SPLINE
SPL {X  -156.240, Y  +354.319, Z    +0.000, E1   +23.538, E3 +157736.290}
SPL {X  -159.137, Y  +372.201, Z    +0.000, E1   +12.017, E3 +157766.128}
SPL {X  -159.858, Y  +382.069, Z    +0.000, E1    +5.945, E3 +157772.645}
SPL {X  -160.000, Y  +389.339, Z    +0.000, E1    +1.101, E3 +157775.807}
SPL {X  -160.000, Y  +395.749, Z    +0.000, E1    -3.722, E3 +157778.413}
SPL {X  -160.000, Y  +403.128, Z    +0.000, E1    -9.899, E3 +157781.717}
SPL {X  -160.000, Y  +411.609, Z    +0.000, E1   -16.851, E3 +157787.038}
SPL {X  -160.000, Y  +429.715, Z    +0.000, E1   -27.376, E3 +157806.401}
SPL {X  -160.000, Y  +449.791, Z    +0.000, E1   -32.145, E3 +157847.638}
SPL {X  -160.000, Y  +454.903, Z    +0.000, E1   -32.134, E3 +157864.943}
SPL {X  -160.000, Y  +460.041, Z    +0.000, E1   -32.144, E3 +157882.296}
SPL {X  -160.000, Y  +465.466, Z    +0.000, E1   -32.152, E3 +157900.614}
SPL {X  -160.000, Y  +471.112, Z    +0.000, E1   -32.154, E3 +157919.702}
SPL {X  -160.000, Y  +476.735, Z    +0.000, E1   -32.156, E3 +157938.693}
SPL {X  -160.000, Y  +482.675, Z    +0.000, E1   -32.169, E3 +157958.742}
SPL {X  -160.000, Y  +488.008, Z    +0.000, E1   -32.144, E3 +157976.788}
SPL {X  -160.000, Y  +493.245, Z    +0.000, E1   -32.159, E3 +157994.497}
SPL {X  -160.000, Y  +498.210, Z    +0.000, E1   -32.128, E3 +158011.331}
SPL {X  -160.000, Y  +503.407, Z    +0.000, E1   -32.165, E3 +158028.835}
SPL {X  -160.000, Y  +509.142, Z    +0.000, E1   -32.157, E3 +158048.231}
SPL {X  -160.000, Y  +514.696, Z    +0.000, E1   -32.156, E3 +158067.011}
SPL {X  -160.000, Y  +520.339, Z    +0.000, E1   -32.159, E3 +158086.083}
SPL {X  -160.000, Y  +525.825, Z    +0.000, E1   -32.148, E3 +158104.647}
SPL {X  -160.000, Y  +530.379, Z    +0.000, E1   -32.130, E3 +158120.075}
SPL {X  -160.000, Y  +535.020, Z    +0.000, E1   -32.146, E3 +158135.721}
SPL {X  -160.000, Y  +540.303, Z    +0.000, E1   -32.158, E3 +158153.546}
SPL {X  -160.000, Y  +545.740, Z    +0.000, E1   -32.155, E3 +158171.939}
SPL {X  -160.000, Y  +550.807, Z    +0.000, E1   -32.147, E3 +158189.062}
SPL {X  -160.000, Y  +555.841, Z    +0.000, E1   -32.148, E3 +158206.101}
SPL {X  -160.000, Y  +561.018, Z    +0.000, E1   -32.143, E3 +158223.630}
SPL {X  -160.000, Y  +566.466, Z    +0.000, E1   -32.153, E3 +158242.048}
SPL {X  -160.000, Y  +571.733, Z    +0.000, E1   -32.135, E3 +158259.885}
SPL {X  -160.000, Y  +576.943, Z    +0.000, E1   -32.148, E3 +158277.481}
SPL {X  -160.000, Y  +582.183, Z    +0.000, E1   -32.140, E3 +158295.206}
SPL {X  -160.000, Y  +587.036, Z    +0.000, E1   -32.141, E3 +158311.577}
SPL {X  -160.000, Y  +591.785, Z    +0.000, E1   -32.144, E3 +158327.601}
SPL {X  -160.000, Y  +596.962, Z    +0.000, E1   -32.161, E3 +158345.087}
SPL {X  -160.000, Y  +601.800, Z    +0.000, E1   -32.134, E3 +158361.484}
SPL {X  -160.000, Y  +606.611, Z    +0.000, E1   -32.156, E3 +158377.699}
SPL {X  -160.000, Y  +611.219, Z    +0.000, E1   -32.131, E3 +158393.312}
SPL {X  -160.000, Y  +616.331, Z    +0.000, E1   -32.174, E3 +158410.510}
SPL {X  -160.000, Y  +621.751, Z    +0.000, E1   -32.150, E3 +158428.853}
SPL {X  -160.000, Y  +626.312, Z    +0.000, E1   -32.145, E3 +158444.258}
SPL {X  -160.000, Y  +630.971, Z    +0.000, E1   -32.155, E3 +158459.987}
SPL {X  -160.000, Y  +635.550, Z    +0.000, E1   -32.137, E3 +158475.513}
SPL {X  -160.000, Y  +640.419, Z    +0.000, E1   -32.158, E3 +158491.951}
SPL {X  -160.000, Y  +645.749, Z    +0.000, E1   -32.151, E3 +158509.976}
SPL {X  -160.000, Y  +650.662, Z    +0.000, E1   -32.150, E3 +158526.547}
SPL {X  -160.000, Y  +655.372, Z    +0.000, E1   -32.145, E3 +158542.494}
SPL {X  -160.000, Y  +660.593, Z    +0.000, E1   -32.163, E3 +158560.112}
SPL {X  -160.000, Y  +665.836, Z    +0.000, E1   -32.154, E3 +158577.828}
SPL {X  -160.000, Y  +670.613, Z    +0.000, E1   -32.138, E3 +158594.039}
SPL {X  -159.954, Y  +675.336, Z    +0.000, E1   -32.135, E3 +158610.047}
SPL {X  -159.758, Y  +680.302, Z    +0.000, E1   -32.108, E3 +158627.062}
SPL {X  -159.416, Y  +685.158, Z    +0.000, E1   -32.039, E3 +158643.873}
SPL {X  -158.953, Y  +689.772, Z    +0.000, E1   -31.965, E3 +158659.972}
SPL {X  -158.363, Y  +694.328, Z    +0.000, E1   -31.871, E3 +158675.985}
SPL {X  -157.606, Y  +699.074, Z    +0.000, E1   -31.756, E3 +158692.828}
SPL {X  -156.791, Y  +703.384, Z    +0.000, E1   -31.607, E3 +158708.278}
SPL {X  -155.792, Y  +707.952, Z    +0.000, E1   -31.465, E3 +158724.725}
SPL {X  -155.149, Y  +710.598, Z    +0.000, E1   -26.183, E3 +158780.185}
ENDSPLINE

SPLINE
SPL {X  -158.679, Y  +692.020, Z    +0.000, E1   -14.212, E3 +158813.861}
SPL {X  -159.747, Y  +680.500, Z    +0.000, E1    -7.378, E3 +158822.238}
SPL {X  -160.000, Y  +671.618, Z    +0.000, E1    -1.592, E3 +158825.853}
SPL {X  -160.000, Y  +666.041, Z    +0.000, E1    +2.615, E3 +158827.819}
SPL {X  -160.000, Y  +661.396, Z    +0.000, E1    +6.484, E3 +158829.492}
SPL {X  -160.000, Y  +653.532, Z    +0.000, E1   +13.136, E3 +158833.613}
SPL {X  -160.000, Y  +631.927, Z    +0.000, E1   +26.832, E3 +158856.379}
SPL {X  -160.000, Y  +610.736, Z    +0.000, E1   +32.114, E3 +158899.049}
SPL {X  -160.000, Y  +605.907, Z    +0.000, E1   +32.114, E3 +158915.397}
SPL {X  -160.000, Y  +601.221, Z    +0.000, E1   +32.108, E3 +158931.264}
SPL {X  -160.000, Y  +596.433, Z    +0.000, E1   +32.120, E3 +158947.447}
SPL {X  -160.000, Y  +592.025, Z    +0.000, E1   +32.104, E3 +158962.371}
SPL {X  -160.000, Y  +587.734, Z    +0.000, E1   +32.110, E3 +158976.891}
SPL {X  -160.000, Y  +583.150, Z    +0.000, E1   +32.111, E3 +158992.419}
SPL {X  -160.000, Y  +579.063, Z    +0.000, E1   +32.085, E3 +159006.320}
SPL {X  -160.000, Y  +574.897, Z    +0.000, E1   +32.110, E3 +159020.372}
SPL {X  -160.000, Y  +570.471, Z    +0.000, E1   +32.093, E3 +159035.386}
SPL {X  -160.000, Y  +566.667, Z    +0.000, E1   +32.086, E3 +159048.300}
SPL {X  -160.000, Y  +562.434, Z    +0.000, E1   +32.097, E3 +159062.610}
SPL {X  -160.000, Y  +557.710, Z    +0.000, E1   +32.104, E3 +159078.593}
SPL {X  -160.000, Y  +553.479, Z    +0.000, E1   +32.081, E3 +159092.963}
SPL {X  -160.000, Y  +547.489, Z    +0.000, E1   +32.181, E3 +159113.081}
SPL {X  -160.000, Y  +541.554, Z    +0.000, E1   +32.092, E3 +159133.318}
SPL {X  -160.000, Y  +537.332, Z    +0.000, E1   +32.092, E3 +159147.616}
SPL {X  -160.000, Y  +533.113, Z    +0.000, E1   +32.090, E3 +159161.912}
SPL {X  -160.000, Y  +528.875, Z    +0.000, E1   +32.090, E3 +159176.256}
SPL {X  -160.000, Y  +524.453, Z    +0.000, E1   +32.104, E3 +159191.180}
SPL {X  -160.000, Y  +520.037, Z    +0.000, E1   +32.096, E3 +159206.122}
SPL {X  -160.000, Y  +514.030, Z    +0.000, E1   +32.182, E3 +159226.318}
SPL {X  -160.000, Y  +508.131, Z    +0.000, E1   +32.099, E3 +159246.422}
SPL {X  -160.000, Y  +504.077, Z    +0.000, E1   +32.094, E3 +159260.145}
SPL {X  -160.000, Y  +494.657, Z    +0.000, E1   +34.509, E3 +159275.008}
SPL {X  -160.000, Y  +491.565, Z    +0.000, E1   +33.823, E3 +159288.915}
SPL {X  -160.000, Y  +489.317, Z    +0.000, E1   +32.894, E3 +159302.260}
SPL {X  -160.000, Y  +486.958, Z    +0.000, E1   +31.703, E3 +159318.032}
SPL {X  -160.000, Y  +484.144, Z    +0.000, E1   +30.999, E3 +159332.455}
SPL {X  -160.000, Y  +479.156, Z    +0.000, E1   +31.035, E3 +159350.021}
SPL {X  -160.000, Y  +474.045, Z    +0.000, E1   +31.015, E3 +159368.112}
SPL {X  -160.000, Y  +468.999, Z    +0.000, E1   +31.021, E3 +159385.937}
SPL {X  -160.000, Y  +464.107, Z    +0.000, E1   +31.012, E3 +159403.238}
SPL {X  -160.000, Y  +459.262, Z    +0.000, E1   +31.016, E3 +159420.345}
SPL {X  -160.000, Y  +454.119, Z    +0.000, E1   +31.026, E3 +159438.494}
SPL {X  -160.000, Y  +448.874, Z    +0.000, E1   +31.019, E3 +159457.050}
SPL {X  -160.000, Y  +443.892, Z    +0.000, E1   +31.019, E3 +159474.638}
SPL {X  -160.000, Y  +438.782, Z    +0.000, E1   +31.022, E3 +159492.712}
SPL {X  -160.000, Y  +433.722, Z    +0.000, E1   +31.007, E3 +159510.656}
SPL {X  -160.000, Y  +428.980, Z    +0.000, E1   +31.004, E3 +159527.413}
SPL {X  -160.000, Y  +424.339, Z    +0.000, E1   +31.006, E3 +159543.788}
SPL {X  -160.000, Y  +419.231, Z    +0.000, E1   +31.030, E3 +159561.781}
SPL {X  -160.000, Y  +414.179, Z    +0.000, E1   +31.008, E3 +159579.678}
SPL {X  -160.000, Y  +409.416, Z    +0.000, E1   +31.023, E3 +159596.462}
SPL {X  -160.000, Y  +403.994, Z    +0.000, E1   +31.033, E3 +159615.617}
SPL {X  -160.000, Y  +399.052, Z    +0.000, E1   +31.010, E3 +159633.085}
SPL {X  -160.000, Y  +394.012, Z    +0.000, E1   +31.036, E3 +159650.874}
SPL {X  -159.999, Y  +388.376, Z    +0.000, E1   +31.028, E3 +159670.804}
SPL {X  -159.897, Y  +383.070, Z    +0.000, E1   +31.010, E3 +159689.642}
SPL {X  -159.656, Y  +378.313, Z    +0.000, E1   +30.961, E3 +159706.734}
SPL {X  -159.237, Y  +373.190, Z    +0.000, E1   +30.917, E3 +159725.234}
SPL {X  -158.628, Y  +367.891, Z    +0.000, E1   +30.812, E3 +159744.620}
SPL {X  -157.915, Y  +363.053, Z    +0.000, E1   +30.689, E3 +159762.487}
SPL {X  -157.216, Y  +359.084, Z    +0.000, E1   +30.550, E3 +159777.289}
SPL {X  -156.248, Y  +354.355, Z    +0.000, E1   +30.460, E3 +159794.902}
SPL {X  -155.629, Y  +351.657, Z    +0.000, E1   +25.972, E3 +159841.330}
ENDSPLINE

SPLINE
SPL {X  -156.240, Y  +354.319, Z    +0.000, E1   +23.538, E3 +159853.938}
SPL {X  -159.137, Y  +372.201, Z    +0.000, E1   +12.017, E3 +159883.775}
SPL {X  -159.858, Y  +382.069, Z    +0.000, E1    +5.945, E3 +159890.293}
SPL {X  -160.000, Y  +389.339, Z    +0.000, E1    +1.101, E3 +159893.455}
SPL {X  -160.000, Y  +395.749, Z    +0.000, E1    -3.722, E3 +159896.060}
SPL {X  -160.000, Y  +403.128, Z    +0.000, E1    -9.899, E3 +159899.364}
SPL {X  -160.000, Y  +411.609, Z    +0.000, E1   -16.851, E3 +159904.685}
SPL {X  -160.000, Y  +429.715, Z    +0.000, E1   -27.376, E3 +159924.049}
SPL {X  -160.000, Y  +449.791, Z    +0.000, E1   -32.145, E3 +159965.286}
SPL {X  -160.000, Y  +454.903, Z    +0.000, E1   -32.134, E3 +159982.590}
SPL {X  -160.000, Y  +460.041, Z    +0.000, E1   -32.144, E3 +159999.943}
SPL {X  -160.000, Y  +465.466, Z    +0.000, E1   -32.152, E3 +160018.261}
SPL {X  -160.000, Y  +471.112, Z    +0.000, E1   -32.154, E3 +160037.350}
SPL {X  -160.000, Y  +476.735, Z    +0.000, E1   -32.156, E3 +160056.340}
SPL {X  -160.000, Y  +482.675, Z    +0.000, E1   -32.169, E3 +160076.389}
SPL {X  -160.000, Y  +488.008, Z    +0.000, E1   -32.144, E3 +160094.436}
SPL {X  -160.000, Y  +493.245, Z    +0.000, E1   -32.159, E3 +160112.144}
SPL {X  -160.000, Y  +498.210, Z    +0.000, E1   -32.128, E3 +160128.979}
SPL {X  -160.000, Y  +503.407, Z    +0.000, E1   -32.165, E3 +160146.482}
SPL {X  -160.000, Y  +509.142, Z    +0.000, E1   -32.157, E3 +160165.878}
SPL {X  -160.000, Y  +514.696, Z    +0.000, E1   -32.156, E3 +160184.658}
SPL {X  -160.000, Y  +520.339, Z    +0.000, E1   -32.159, E3 +160203.731}
SPL {X  -160.000, Y  +525.825, Z    +0.000, E1   -32.148, E3 +160222.294}
SPL {X  -160.000, Y  +530.379, Z    +0.000, E1   -32.130, E3 +160237.722}
SPL {X  -160.000, Y  +535.020, Z    +0.000, E1   -32.146, E3 +160253.368}
SPL {X  -160.000, Y  +540.303, Z    +0.000, E1   -32.158, E3 +160271.194}
SPL {X  -160.000, Y  +545.740, Z    +0.000, E1   -32.155, E3 +160289.586}
SPL {X  -160.000, Y  +550.807, Z    +0.000, E1   -32.147, E3 +160306.709}
SPL {X  -160.000, Y  +555.841, Z    +0.000, E1   -32.148, E3 +160323.748}
SPL {X  -160.000, Y  +561.018, Z    +0.000, E1   -32.143, E3 +160341.277}
SPL {X  -160.000, Y  +566.466, Z    +0.000, E1   -32.153, E3 +160359.695}
SPL {X  -160.000, Y  +571.733, Z    +0.000, E1   -32.135, E3 +160377.532}
SPL {X  -160.000, Y  +576.943, Z    +0.000, E1   -32.148, E3 +160395.129}
SPL {X  -160.000, Y  +582.183, Z    +0.000, E1   -32.140, E3 +160412.854}
SPL {X  -160.000, Y  +587.036, Z    +0.000, E1   -32.141, E3 +160429.224}
SPL {X  -160.000, Y  +591.785, Z    +0.000, E1   -32.144, E3 +160445.248}
SPL {X  -160.000, Y  +596.962, Z    +0.000, E1   -32.161, E3 +160462.735}
SPL {X  -160.000, Y  +601.800, Z    +0.000, E1   -32.134, E3 +160479.132}
SPL {X  -160.000, Y  +606.611, Z    +0.000, E1   -32.156, E3 +160495.346}
SPL {X  -160.000, Y  +611.219, Z    +0.000, E1   -32.131, E3 +160510.960}
SPL {X  -160.000, Y  +616.331, Z    +0.000, E1   -32.174, E3 +160528.157}
SPL {X  -160.000, Y  +621.751, Z    +0.000, E1   -32.150, E3 +160546.500}
SPL {X  -160.000, Y  +626.312, Z    +0.000, E1   -32.145, E3 +160561.906}
SPL {X  -160.000, Y  +630.971, Z    +0.000, E1   -32.155, E3 +160577.634}
SPL {X  -160.000, Y  +635.550, Z    +0.000, E1   -32.137, E3 +160593.160}
SPL {X  -160.000, Y  +640.419, Z    +0.000, E1   -32.158, E3 +160609.598}
SPL {X  -160.000, Y  +645.749, Z    +0.000, E1   -32.151, E3 +160627.623}
SPL {X  -160.000, Y  +650.662, Z    +0.000, E1   -32.150, E3 +160644.194}
SPL {X  -160.000, Y  +655.372, Z    +0.000, E1   -32.145, E3 +160660.141}
SPL {X  -160.000, Y  +660.593, Z    +0.000, E1   -32.163, E3 +160677.759}
SPL {X  -160.000, Y  +665.836, Z    +0.000, E1   -32.154, E3 +160695.476}
SPL {X  -160.000, Y  +670.613, Z    +0.000, E1   -32.138, E3 +160711.686}
SPL {X  -159.954, Y  +675.336, Z    +0.000, E1   -32.135, E3 +160727.694}
SPL {X  -159.758, Y  +680.302, Z    +0.000, E1   -32.108, E3 +160744.709}
SPL {X  -159.416, Y  +685.158, Z    +0.000, E1   -32.039, E3 +160761.520}
SPL {X  -158.953, Y  +689.772, Z    +0.000, E1   -31.965, E3 +160777.619}
SPL {X  -158.363, Y  +694.328, Z    +0.000, E1   -31.871, E3 +160793.632}
SPL {X  -157.606, Y  +699.074, Z    +0.000, E1   -31.756, E3 +160810.475}
SPL {X  -156.791, Y  +703.384, Z    +0.000, E1   -31.607, E3 +160825.926}
SPL {X  -155.792, Y  +707.952, Z    +0.000, E1   -31.465, E3 +160842.372}
SPL {X  -155.149, Y  +710.598, Z    +0.000, E1   -26.183, E3 +160897.832}
ENDSPLINE

SPLINE
SPL {X  -158.679, Y  +692.020, Z    +0.000, E1   -14.212, E3 +160931.508}
SPL {X  -159.747, Y  +680.500, Z    +0.000, E1    -7.378, E3 +160939.886}
SPL {X  -160.000, Y  +671.618, Z    +0.000, E1    -1.592, E3 +160943.500}
SPL {X  -160.000, Y  +666.041, Z    +0.000, E1    +2.615, E3 +160945.467}
SPL {X  -160.000, Y  +661.396, Z    +0.000, E1    +6.484, E3 +160947.140}
SPL {X  -160.000, Y  +653.532, Z    +0.000, E1   +13.136, E3 +160951.260}
SPL {X  -160.000, Y  +631.927, Z    +0.000, E1   +26.832, E3 +160974.027}
SPL {X  -160.000, Y  +610.736, Z    +0.000, E1   +32.114, E3 +161016.696}
SPL {X  -160.000, Y  +605.907, Z    +0.000, E1   +32.114, E3 +161033.044}
SPL {X  -160.000, Y  +601.221, Z    +0.000, E1   +32.108, E3 +161048.912}
SPL {X  -160.000, Y  +596.433, Z    +0.000, E1   +32.120, E3 +161065.094}
SPL {X  -160.000, Y  +592.025, Z    +0.000, E1   +32.104, E3 +161080.018}
SPL {X  -160.000, Y  +587.734, Z    +0.000, E1   +32.110, E3 +161094.539}
SPL {X  -160.000, Y  +583.150, Z    +0.000, E1   +32.111, E3 +161110.066}
SPL {X  -160.000, Y  +579.063, Z    +0.000, E1   +32.085, E3 +161123.968}
SPL {X  -160.000, Y  +574.897, Z    +0.000, E1   +32.110, E3 +161138.019}
SPL {X  -160.000, Y  +570.471, Z    +0.000, E1   +32.093, E3 +161153.033}
SPL {X  -160.000, Y  +566.667, Z    +0.000, E1   +32.086, E3 +161165.948}
SPL {X  -160.000, Y  +562.434, Z    +0.000, E1   +32.097, E3 +161180.257}
SPL {X  -160.000, Y  +557.710, Z    +0.000, E1   +32.104, E3 +161196.241}
SPL {X  -160.000, Y  +553.479, Z    +0.000, E1   +32.081, E3 +161210.610}
SPL {X  -160.000, Y  +547.489, Z    +0.000, E1   +32.181, E3 +161230.729}
SPL {X  -160.000, Y  +541.554, Z    +0.000, E1   +32.092, E3 +161250.966}
SPL {X  -160.000, Y  +537.332, Z    +0.000, E1   +32.092, E3 +161265.263}
SPL {X  -160.000, Y  +533.113, Z    +0.000, E1   +32.090, E3 +161279.560}
SPL {X  -160.000, Y  +528.875, Z    +0.000, E1   +32.090, E3 +161293.903}
SPL {X  -160.000, Y  +524.453, Z    +0.000, E1   +32.104, E3 +161308.827}
SPL {X  -160.000, Y  +520.037, Z    +0.000, E1   +32.096, E3 +161323.769}
SPL {X  -160.000, Y  +514.030, Z    +0.000, E1   +32.182, E3 +161343.965}
SPL {X  -160.000, Y  +508.131, Z    +0.000, E1   +32.099, E3 +161364.069}
SPL {X  -160.000, Y  +504.077, Z    +0.000, E1   +32.094, E3 +161377.792}
SPL {X  -160.000, Y  +494.657, Z    +0.000, E1   +34.509, E3 +161392.655}
SPL {X  -160.000, Y  +491.565, Z    +0.000, E1   +33.823, E3 +161406.563}
SPL {X  -160.000, Y  +489.317, Z    +0.000, E1   +32.894, E3 +161419.907}
SPL {X  -160.000, Y  +486.958, Z    +0.000, E1   +31.703, E3 +161435.679}
SPL {X  -160.000, Y  +484.144, Z    +0.000, E1   +30.999, E3 +161450.102}
SPL {X  -160.000, Y  +479.156, Z    +0.000, E1   +31.035, E3 +161467.668}
SPL {X  -160.000, Y  +474.045, Z    +0.000, E1   +31.015, E3 +161485.760}
SPL {X  -160.000, Y  +468.999, Z    +0.000, E1   +31.021, E3 +161503.585}
SPL {X  -160.000, Y  +464.107, Z    +0.000, E1   +31.012, E3 +161520.885}
SPL {X  -160.000, Y  +459.262, Z    +0.000, E1   +31.016, E3 +161537.992}
SPL {X  -160.000, Y  +454.119, Z    +0.000, E1   +31.026, E3 +161556.141}
SPL {X  -160.000, Y  +448.874, Z    +0.000, E1   +31.019, E3 +161574.697}
SPL {X  -160.000, Y  +443.892, Z    +0.000, E1   +31.019, E3 +161592.285}
SPL {X  -160.000, Y  +438.782, Z    +0.000, E1   +31.022, E3 +161610.360}
SPL {X  -160.000, Y  +433.722, Z    +0.000, E1   +31.007, E3 +161628.303}
SPL {X  -160.000, Y  +428.980, Z    +0.000, E1   +31.004, E3 +161645.061}
SPL {X  -160.000, Y  +424.339, Z    +0.000, E1   +31.006, E3 +161661.435}
SPL {X  -160.000, Y  +419.231, Z    +0.000, E1   +31.030, E3 +161679.428}
SPL {X  -160.000, Y  +414.179, Z    +0.000, E1   +31.008, E3 +161697.326}
SPL {X  -160.000, Y  +409.416, Z    +0.000, E1   +31.023, E3 +161714.109}
SPL {X  -160.000, Y  +403.994, Z    +0.000, E1   +31.033, E3 +161733.264}
SPL {X  -160.000, Y  +399.052, Z    +0.000, E1   +31.010, E3 +161750.732}
SPL {X  -160.000, Y  +394.012, Z    +0.000, E1   +31.036, E3 +161768.521}
SPL {X  -159.999, Y  +388.376, Z    +0.000, E1   +31.028, E3 +161788.451}
SPL {X  -159.897, Y  +383.070, Z    +0.000, E1   +31.010, E3 +161807.289}
SPL {X  -159.656, Y  +378.313, Z    +0.000, E1   +30.961, E3 +161824.381}
SPL {X  -159.237, Y  +373.190, Z    +0.000, E1   +30.917, E3 +161842.881}
SPL {X  -158.628, Y  +367.891, Z    +0.000, E1   +30.812, E3 +161862.267}
SPL {X  -157.915, Y  +363.053, Z    +0.000, E1   +30.689, E3 +161880.134}
SPL {X  -157.216, Y  +359.084, Z    +0.000, E1   +30.550, E3 +161894.937}
SPL {X  -156.248, Y  +354.355, Z    +0.000, E1   +30.460, E3 +161912.549}
SPL {X  -155.629, Y  +351.657, Z    +0.000, E1   +25.972, E3 +161958.977}
ENDSPLINE

SPLINE
SPL {X  -156.240, Y  +354.319, Z    +0.000, E1   +23.538, E3 +161971.585}
SPL {X  -159.137, Y  +372.201, Z    +0.000, E1   +12.017, E3 +162001.422}
SPL {X  -159.858, Y  +382.069, Z    +0.000, E1    +5.945, E3 +162007.940}
SPL {X  -160.000, Y  +389.339, Z    +0.000, E1    +1.101, E3 +162011.102}
SPL {X  -160.000, Y  +395.749, Z    +0.000, E1    -3.722, E3 +162013.707}
SPL {X  -160.000, Y  +403.128, Z    +0.000, E1    -9.899, E3 +162017.012}
SPL {X  -160.000, Y  +411.609, Z    +0.000, E1   -16.851, E3 +162022.332}
SPL {X  -160.000, Y  +429.715, Z    +0.000, E1   -27.376, E3 +162041.696}
SPL {X  -160.000, Y  +449.791, Z    +0.000, E1   -32.145, E3 +162082.933}
SPL {X  -160.000, Y  +454.903, Z    +0.000, E1   -32.134, E3 +162100.237}
SPL {X  -160.000, Y  +460.041, Z    +0.000, E1   -32.144, E3 +162117.591}
SPL {X  -160.000, Y  +465.466, Z    +0.000, E1   -32.152, E3 +162135.909}
SPL {X  -160.000, Y  +471.112, Z    +0.000, E1   -32.154, E3 +162154.997}
SPL {X  -160.000, Y  +476.735, Z    +0.000, E1   -32.156, E3 +162173.988}
SPL {X  -160.000, Y  +482.675, Z    +0.000, E1   -32.169, E3 +162194.037}
SPL {X  -160.000, Y  +488.008, Z    +0.000, E1   -32.144, E3 +162212.083}
SPL {X  -160.000, Y  +493.245, Z    +0.000, E1   -32.159, E3 +162229.791}
SPL {X  -160.000, Y  +498.210, Z    +0.000, E1   -32.128, E3 +162246.626}
SPL {X  -160.000, Y  +503.407, Z    +0.000, E1   -32.165, E3 +162264.130}
SPL {X  -160.000, Y  +509.142, Z    +0.000, E1   -32.157, E3 +162283.525}
SPL {X  -160.000, Y  +514.696, Z    +0.000, E1   -32.156, E3 +162302.306}
SPL {X  -160.000, Y  +520.339, Z    +0.000, E1   -32.159, E3 +162321.378}
SPL {X  -160.000, Y  +525.825, Z    +0.000, E1   -32.148, E3 +162339.941}
SPL {X  -160.000, Y  +530.379, Z    +0.000, E1   -32.130, E3 +162355.370}
SPL {X  -160.000, Y  +535.020, Z    +0.000, E1   -32.146, E3 +162371.016}
SPL {X  -160.000, Y  +540.303, Z    +0.000, E1   -32.158, E3 +162388.841}
SPL {X  -160.000, Y  +545.740, Z    +0.000, E1   -32.155, E3 +162407.234}
SPL {X  -160.000, Y  +550.807, Z    +0.000, E1   -32.147, E3 +162424.356}
SPL {X  -160.000, Y  +555.841, Z    +0.000, E1   -32.148, E3 +162441.396}
SPL {X  -160.000, Y  +561.018, Z    +0.000, E1   -32.143, E3 +162458.924}
SPL {X  -160.000, Y  +566.466, Z    +0.000, E1   -32.153, E3 +162477.343}
SPL {X  -160.000, Y  +571.733, Z    +0.000, E1   -32.135, E3 +162495.179}
SPL {X  -160.000, Y  +576.943, Z    +0.000, E1   -32.148, E3 +162512.776}
SPL {X  -160.000, Y  +582.183, Z    +0.000, E1   -32.140, E3 +162530.501}
SPL {X  -160.000, Y  +587.036, Z    +0.000, E1   -32.141, E3 +162546.872}
SPL {X  -160.000, Y  +591.785, Z    +0.000, E1   -32.144, E3 +162562.895}
SPL {X  -160.000, Y  +596.962, Z    +0.000, E1   -32.161, E3 +162580.382}
SPL {X  -160.000, Y  +601.800, Z    +0.000, E1   -32.134, E3 +162596.779}
SPL {X  -160.000, Y  +606.611, Z    +0.000, E1   -32.156, E3 +162612.993}
SPL {X  -160.000, Y  +611.219, Z    +0.000, E1   -32.131, E3 +162628.607}
SPL {X  -160.000, Y  +616.331, Z    +0.000, E1   -32.174, E3 +162645.805}
SPL {X  -160.000, Y  +621.751, Z    +0.000, E1   -32.150, E3 +162664.147}
SPL {X  -160.000, Y  +626.312, Z    +0.000, E1   -32.145, E3 +162679.553}
SPL {X  -160.000, Y  +630.971, Z    +0.000, E1   -32.155, E3 +162695.281}
SPL {X  -160.000, Y  +635.550, Z    +0.000, E1   -32.137, E3 +162710.807}
SPL {X  -160.000, Y  +640.419, Z    +0.000, E1   -32.158, E3 +162727.245}
SPL {X  -160.000, Y  +645.749, Z    +0.000, E1   -32.151, E3 +162745.271}
SPL {X  -160.000, Y  +650.662, Z    +0.000, E1   -32.150, E3 +162761.842}
SPL {X  -160.000, Y  +655.372, Z    +0.000, E1   -32.145, E3 +162777.789}
SPL {X  -160.000, Y  +660.593, Z    +0.000, E1   -32.163, E3 +162795.406}
SPL {X  -160.000, Y  +665.836, Z    +0.000, E1   -32.154, E3 +162813.123}
SPL {X  -160.000, Y  +670.613, Z    +0.000, E1   -32.138, E3 +162829.333}
SPL {X  -159.954, Y  +675.336, Z    +0.000, E1   -32.135, E3 +162845.341}
SPL {X  -159.758, Y  +680.302, Z    +0.000, E1   -32.108, E3 +162862.356}
SPL {X  -159.416, Y  +685.158, Z    +0.000, E1   -32.039, E3 +162879.167}
SPL {X  -158.953, Y  +689.772, Z    +0.000, E1   -31.965, E3 +162895.267}
SPL {X  -158.363, Y  +694.328, Z    +0.000, E1   -31.871, E3 +162911.279}
SPL {X  -157.606, Y  +699.074, Z    +0.000, E1   -31.756, E3 +162928.123}
SPL {X  -156.791, Y  +703.384, Z    +0.000, E1   -31.607, E3 +162943.573}
SPL {X  -155.792, Y  +707.952, Z    +0.000, E1   -31.465, E3 +162960.019}
SPL {X  -155.149, Y  +710.598, Z    +0.000, E1   -26.183, E3 +163015.479}
ENDSPLINE

SPLINE
SPL {X  -158.679, Y  +692.020, Z    +0.000, E1   -14.212, E3 +163049.155}
SPL {X  -159.747, Y  +680.500, Z    +0.000, E1    -7.378, E3 +163057.533}
SPL {X  -160.000, Y  +671.618, Z    +0.000, E1    -1.592, E3 +163061.147}
SPL {X  -160.000, Y  +666.041, Z    +0.000, E1    +2.615, E3 +163063.114}
SPL {X  -160.000, Y  +661.396, Z    +0.000, E1    +6.484, E3 +163064.787}
SPL {X  -160.000, Y  +653.532, Z    +0.000, E1   +13.136, E3 +163068.907}
SPL {X  -160.000, Y  +631.927, Z    +0.000, E1   +26.832, E3 +163091.674}
SPL {X  -160.000, Y  +610.736, Z    +0.000, E1   +32.114, E3 +163134.343}
SPL {X  -160.000, Y  +605.907, Z    +0.000, E1   +32.114, E3 +163150.692}
SPL {X  -160.000, Y  +601.221, Z    +0.000, E1   +32.108, E3 +163166.559}
SPL {X  -160.000, Y  +596.433, Z    +0.000, E1   +32.120, E3 +163182.741}
SPL {X  -160.000, Y  +592.025, Z    +0.000, E1   +32.104, E3 +163197.666}
SPL {X  -160.000, Y  +587.734, Z    +0.000, E1   +32.110, E3 +163212.186}
SPL {X  -160.000, Y  +583.150, Z    +0.000, E1   +32.111, E3 +163227.714}
SPL {X  -160.000, Y  +579.063, Z    +0.000, E1   +32.085, E3 +163241.615}
SPL {X  -160.000, Y  +574.897, Z    +0.000, E1   +32.110, E3 +163255.666}
SPL {X  -160.000, Y  +570.471, Z    +0.000, E1   +32.093, E3 +163270.681}
SPL {X  -160.000, Y  +566.667, Z    +0.000, E1   +32.086, E3 +163283.595}
SPL {X  -160.000, Y  +562.434, Z    +0.000, E1   +32.097, E3 +163297.905}
SPL {X  -160.000, Y  +557.710, Z    +0.000, E1   +32.104, E3 +163313.888}
SPL {X  -160.000, Y  +553.479, Z    +0.000, E1   +32.081, E3 +163328.257}
SPL {X  -160.000, Y  +547.489, Z    +0.000, E1   +32.181, E3 +163348.376}
SPL {X  -160.000, Y  +541.554, Z    +0.000, E1   +32.092, E3 +163368.613}
SPL {X  -160.000, Y  +537.332, Z    +0.000, E1   +32.092, E3 +163382.910}
SPL {X  -160.000, Y  +533.113, Z    +0.000, E1   +32.090, E3 +163397.207}
SPL {X  -160.000, Y  +528.875, Z    +0.000, E1   +32.090, E3 +163411.550}
SPL {X  -160.000, Y  +524.453, Z    +0.000, E1   +32.104, E3 +163426.474}
SPL {X  -160.000, Y  +520.037, Z    +0.000, E1   +32.096, E3 +163441.416}
SPL {X  -160.000, Y  +514.030, Z    +0.000, E1   +32.182, E3 +163461.612}
SPL {X  -160.000, Y  +508.131, Z    +0.000, E1   +32.099, E3 +163481.717}
SPL {X  -160.000, Y  +504.077, Z    +0.000, E1   +32.094, E3 +163495.440}
SPL {X  -160.000, Y  +494.657, Z    +0.000, E1   +34.509, E3 +163510.303}
SPL {X  -160.000, Y  +491.565, Z    +0.000, E1   +33.823, E3 +163524.210}
SPL {X  -160.000, Y  +489.317, Z    +0.000, E1   +32.894, E3 +163537.555}
SPL {X  -160.000, Y  +486.958, Z    +0.000, E1   +31.703, E3 +163553.326}
SPL {X  -160.000, Y  +484.144, Z    +0.000, E1   +30.999, E3 +163567.749}
SPL {X  -160.000, Y  +479.156, Z    +0.000, E1   +31.035, E3 +163585.315}
SPL {X  -160.000, Y  +474.045, Z    +0.000, E1   +31.015, E3 +163603.407}
SPL {X  -160.000, Y  +468.999, Z    +0.000, E1   +31.021, E3 +163621.232}
SPL {X  -160.000, Y  +464.107, Z    +0.000, E1   +31.012, E3 +163638.532}
SPL {X  -160.000, Y  +459.262, Z    +0.000, E1   +31.016, E3 +163655.639}
SPL {X  -160.000, Y  +454.119, Z    +0.000, E1   +31.026, E3 +163673.789}
SPL {X  -160.000, Y  +448.874, Z    +0.000, E1   +31.019, E3 +163692.344}
SPL {X  -160.000, Y  +443.892, Z    +0.000, E1   +31.019, E3 +163709.933}
SPL {X  -160.000, Y  +438.782, Z    +0.000, E1   +31.022, E3 +163728.007}
SPL {X  -160.000, Y  +433.722, Z    +0.000, E1   +31.007, E3 +163745.951}
SPL {X  -160.000, Y  +428.980, Z    +0.000, E1   +31.004, E3 +163762.708}
SPL {X  -160.000, Y  +424.339, Z    +0.000, E1   +31.006, E3 +163779.082}
SPL {X  -160.000, Y  +419.231, Z    +0.000, E1   +31.030, E3 +163797.076}
SPL {X  -160.000, Y  +414.179, Z    +0.000, E1   +31.008, E3 +163814.973}
SPL {X  -160.000, Y  +409.416, Z    +0.000, E1   +31.023, E3 +163831.756}
SPL {X  -160.000, Y  +403.994, Z    +0.000, E1   +31.033, E3 +163850.912}
SPL {X  -160.000, Y  +399.052, Z    +0.000, E1   +31.010, E3 +163868.380}
SPL {X  -160.000, Y  +394.012, Z    +0.000, E1   +31.036, E3 +163886.168}
SPL {X  -159.999, Y  +388.376, Z    +0.000, E1   +31.028, E3 +163906.098}
SPL {X  -159.897, Y  +383.070, Z    +0.000, E1   +31.010, E3 +163924.936}
SPL {X  -159.656, Y  +378.313, Z    +0.000, E1   +30.961, E3 +163942.028}
SPL {X  -159.237, Y  +373.190, Z    +0.000, E1   +30.917, E3 +163960.529}
SPL {X  -158.628, Y  +367.891, Z    +0.000, E1   +30.812, E3 +163979.914}
SPL {X  -157.915, Y  +363.053, Z    +0.000, E1   +30.689, E3 +163997.781}
SPL {X  -157.216, Y  +359.084, Z    +0.000, E1   +30.550, E3 +164012.584}
SPL {X  -156.248, Y  +354.355, Z    +0.000, E1   +30.460, E3 +164030.196}
SPL {X  -155.629, Y  +351.657, Z    +0.000, E1   +25.972, E3 +164076.625}
ENDSPLINE

SPLINE
SPL {X  -156.240, Y  +354.319, Z    +0.000, E1   +23.538, E3 +164089.232}
SPL {X  -159.137, Y  +372.201, Z    +0.000, E1   +12.017, E3 +164119.069}
SPL {X  -159.858, Y  +382.069, Z    +0.000, E1    +5.945, E3 +164125.587}
SPL {X  -160.000, Y  +389.339, Z    +0.000, E1    +1.101, E3 +164128.749}
SPL {X  -160.000, Y  +395.749, Z    +0.000, E1    -3.722, E3 +164131.355}
SPL {X  -160.000, Y  +403.128, Z    +0.000, E1    -9.899, E3 +164134.659}
SPL {X  -160.000, Y  +411.609, Z    +0.000, E1   -16.851, E3 +164139.980}
SPL {X  -160.000, Y  +429.715, Z    +0.000, E1   -27.376, E3 +164159.343}
SPL {X  -160.000, Y  +449.791, Z    +0.000, E1   -32.145, E3 +164200.580}
SPL {X  -160.000, Y  +454.903, Z    +0.000, E1   -32.134, E3 +164217.885}
SPL {X  -160.000, Y  +460.041, Z    +0.000, E1   -32.144, E3 +164235.238}
SPL {X  -160.000, Y  +465.466, Z    +0.000, E1   -32.152, E3 +164253.556}
SPL {X  -160.000, Y  +471.112, Z    +0.000, E1   -32.154, E3 +164272.644}
SPL {X  -160.000, Y  +476.735, Z    +0.000, E1   -32.156, E3 +164291.635}
SPL {X  -160.000, Y  +482.675, Z    +0.000, E1   -32.169, E3 +164311.684}
SPL {X  -160.000, Y  +488.008, Z    +0.000, E1   -32.144, E3 +164329.730}
SPL {X  -160.000, Y  +493.245, Z    +0.000, E1   -32.159, E3 +164347.439}
SPL {X  -160.000, Y  +498.210, Z    +0.000, E1   -32.128, E3 +164364.273}
SPL {X  -160.000, Y  +503.407, Z    +0.000, E1   -32.165, E3 +164381.777}
SPL {X  -160.000, Y  +509.142, Z    +0.000, E1   -32.157, E3 +164401.173}
SPL {X  -160.000, Y  +514.696, Z    +0.000, E1   -32.156, E3 +164419.953}
SPL {X  -160.000, Y  +520.339, Z    +0.000, E1   -32.159, E3 +164439.025}
SPL {X  -160.000, Y  +525.825, Z    +0.000, E1   -32.148, E3 +164457.589}
SPL {X  -160.000, Y  +530.379, Z    +0.000, E1   -32.130, E3 +164473.017}
SPL {X  -160.000, Y  +535.020, Z    +0.000, E1   -32.146, E3 +164488.663}
SPL {X  -160.000, Y  +540.303, Z    +0.000, E1   -32.158, E3 +164506.488}
SPL {X  -160.000, Y  +545.740, Z    +0.000, E1   -32.155, E3 +164524.881}
SPL {X  -160.000, Y  +550.807, Z    +0.000, E1   -32.147, E3 +164542.004}
SPL {X  -160.000, Y  +555.841, Z    +0.000, E1   -32.148, E3 +164559.043}
SPL {X  -160.000, Y  +561.018, Z    +0.000, E1   -32.143, E3 +164576.572}
SPL {X  -160.000, Y  +566.466, Z    +0.000, E1   -32.153, E3 +164594.990}
SPL {X  -160.000, Y  +571.733, Z    +0.000, E1   -32.135, E3 +164612.827}
SPL {X  -160.000, Y  +576.943, Z    +0.000, E1   -32.148, E3 +164630.423}
SPL {X  -160.000, Y  +582.183, Z    +0.000, E1   -32.140, E3 +164648.148}
SPL {X  -160.000, Y  +587.036, Z    +0.000, E1   -32.141, E3 +164664.519}
SPL {X  -160.000, Y  +591.785, Z    +0.000, E1   -32.144, E3 +164680.543}
SPL {X  -160.000, Y  +596.962, Z    +0.000, E1   -32.161, E3 +164698.029}
SPL {X  -160.000, Y  +601.800, Z    +0.000, E1   -32.134, E3 +164714.426}
SPL {X  -160.000, Y  +606.611, Z    +0.000, E1   -32.156, E3 +164730.641}
SPL {X  -160.000, Y  +611.219, Z    +0.000, E1   -32.131, E3 +164746.254}
SPL {X  -160.000, Y  +616.331, Z    +0.000, E1   -32.174, E3 +164763.452}
SPL {X  -160.000, Y  +621.751, Z    +0.000, E1   -32.150, E3 +164781.795}
SPL {X  -160.000, Y  +626.312, Z    +0.000, E1   -32.145, E3 +164797.200}
SPL {X  -160.000, Y  +630.971, Z    +0.000, E1   -32.155, E3 +164812.929}
SPL {X  -160.000, Y  +635.550, Z    +0.000, E1   -32.137, E3 +164828.454}
SPL {X  -160.000, Y  +640.419, Z    +0.000, E1   -32.158, E3 +164844.892}
SPL {X  -160.000, Y  +645.749, Z    +0.000, E1   -32.151, E3 +164862.918}
SPL {X  -160.000, Y  +650.662, Z    +0.000, E1   -32.150, E3 +164879.489}
SPL {X  -160.000, Y  +655.372, Z    +0.000, E1   -32.145, E3 +164895.436}
SPL {X  -160.000, Y  +660.593, Z    +0.000, E1   -32.163, E3 +164913.054}
SPL {X  -160.000, Y  +665.836, Z    +0.000, E1   -32.154, E3 +164930.770}
SPL {X  -160.000, Y  +670.613, Z    +0.000, E1   -32.138, E3 +164946.980}
SPL {X  -159.954, Y  +675.336, Z    +0.000, E1   -32.135, E3 +164962.989}
SPL {X  -159.758, Y  +680.302, Z    +0.000, E1   -32.108, E3 +164980.003}
SPL {X  -159.416, Y  +685.158, Z    +0.000, E1   -32.039, E3 +164996.815}
SPL {X  -158.953, Y  +689.772, Z    +0.000, E1   -31.965, E3 +165012.914}
SPL {X  -158.363, Y  +694.328, Z    +0.000, E1   -31.871, E3 +165028.927}
SPL {X  -157.606, Y  +699.074, Z    +0.000, E1   -31.756, E3 +165045.770}
SPL {X  -156.791, Y  +703.384, Z    +0.000, E1   -31.607, E3 +165061.220}
SPL {X  -155.792, Y  +707.952, Z    +0.000, E1   -31.465, E3 +165077.667}
SPL {X  -155.149, Y  +710.598, Z    +0.000, E1   -26.183, E3 +165133.126}
ENDSPLINE

SPLINE
SPL {X  -158.679, Y  +692.020, Z    +0.000, E1   -14.212, E3 +165166.803}
SPL {X  -159.747, Y  +680.500, Z    +0.000, E1    -7.378, E3 +165175.180}
SPL {X  -160.000, Y  +671.618, Z    +0.000, E1    -1.592, E3 +165178.795}
SPL {X  -160.000, Y  +666.041, Z    +0.000, E1    +2.615, E3 +165180.761}
SPL {X  -160.000, Y  +661.396, Z    +0.000, E1    +6.484, E3 +165182.434}
SPL {X  -160.000, Y  +653.532, Z    +0.000, E1   +13.136, E3 +165186.554}
SPL {X  -160.000, Y  +631.927, Z    +0.000, E1   +26.832, E3 +165209.321}
SPL {X  -160.000, Y  +610.736, Z    +0.000, E1   +32.114, E3 +165251.991}
SPL {X  -160.000, Y  +605.907, Z    +0.000, E1   +32.114, E3 +165268.339}
SPL {X  -160.000, Y  +601.221, Z    +0.000, E1   +32.108, E3 +165284.206}
SPL {X  -160.000, Y  +596.433, Z    +0.000, E1   +32.120, E3 +165300.388}
SPL {X  -160.000, Y  +592.025, Z    +0.000, E1   +32.104, E3 +165315.313}
SPL {X  -160.000, Y  +587.734, Z    +0.000, E1   +32.110, E3 +165329.833}
SPL {X  -160.000, Y  +583.150, Z    +0.000, E1   +32.111, E3 +165345.361}
SPL {X  -160.000, Y  +579.063, Z    +0.000, E1   +32.085, E3 +165359.262}
SPL {X  -160.000, Y  +574.897, Z    +0.000, E1   +32.110, E3 +165373.314}
SPL {X  -160.000, Y  +570.471, Z    +0.000, E1   +32.093, E3 +165388.328}
SPL {X  -160.000, Y  +566.667, Z    +0.000, E1   +32.086, E3 +165401.242}
SPL {X  -160.000, Y  +562.434, Z    +0.000, E1   +32.097, E3 +165415.552}
SPL {X  -160.000, Y  +557.710, Z    +0.000, E1   +32.104, E3 +165431.535}
SPL {X  -160.000, Y  +553.479, Z    +0.000, E1   +32.081, E3 +165445.905}
SPL {X  -160.000, Y  +547.489, Z    +0.000, E1   +32.181, E3 +165466.023}
SPL {X  -160.000, Y  +541.554, Z    +0.000, E1   +32.092, E3 +165486.260}
SPL {X  -160.000, Y  +537.332, Z    +0.000, E1   +32.092, E3 +165500.557}
SPL {X  -160.000, Y  +533.113, Z    +0.000, E1   +32.090, E3 +165514.854}
SPL {X  -160.000, Y  +528.875, Z    +0.000, E1   +32.090, E3 +165529.198}
SPL {X  -160.000, Y  +524.453, Z    +0.000, E1   +32.104, E3 +165544.121}
SPL {X  -160.000, Y  +520.037, Z    +0.000, E1   +32.096, E3 +165559.064}
SPL {X  -160.000, Y  +514.030, Z    +0.000, E1   +32.182, E3 +165579.260}
SPL {X  -160.000, Y  +508.131, Z    +0.000, E1   +32.099, E3 +165599.364}
SPL {X  -160.000, Y  +504.077, Z    +0.000, E1   +32.094, E3 +165613.087}
SPL {X  -160.000, Y  +494.657, Z    +0.000, E1   +34.509, E3 +165627.950}
SPL {X  -160.000, Y  +491.565, Z    +0.000, E1   +33.823, E3 +165641.857}
SPL {X  -160.000, Y  +489.317, Z    +0.000, E1   +32.894, E3 +165655.202}
SPL {X  -160.000, Y  +486.958, Z    +0.000, E1   +31.703, E3 +165670.974}
SPL {X  -160.000, Y  +484.144, Z    +0.000, E1   +30.999, E3 +165685.396}
SPL {X  -160.000, Y  +479.156, Z    +0.000, E1   +31.035, E3 +165702.962}
SPL {X  -160.000, Y  +474.045, Z    +0.000, E1   +31.015, E3 +165721.054}
SPL {X  -160.000, Y  +468.999, Z    +0.000, E1   +31.021, E3 +165738.879}
SPL {X  -160.000, Y  +464.107, Z    +0.000, E1   +31.012, E3 +165756.179}
SPL {X  -160.000, Y  +459.262, Z    +0.000, E1   +31.016, E3 +165773.286}
SPL {X  -160.000, Y  +454.119, Z    +0.000, E1   +31.026, E3 +165791.436}
SPL {X  -160.000, Y  +448.874, Z    +0.000, E1   +31.019, E3 +165809.992}
SPL {X  -160.000, Y  +443.892, Z    +0.000, E1   +31.019, E3 +165827.580}
SPL {X  -160.000, Y  +438.782, Z    +0.000, E1   +31.022, E3 +165845.654}
SPL {X  -160.000, Y  +433.722, Z    +0.000, E1   +31.007, E3 +165863.598}
SPL {X  -160.000, Y  +428.980, Z    +0.000, E1   +31.004, E3 +165880.355}
SPL {X  -160.000, Y  +424.339, Z    +0.000, E1   +31.006, E3 +165896.729}
SPL {X  -160.000, Y  +419.231, Z    +0.000, E1   +31.030, E3 +165914.723}
SPL {X  -160.000, Y  +414.179, Z    +0.000, E1   +31.008, E3 +165932.620}
SPL {X  -160.000, Y  +409.416, Z    +0.000, E1   +31.023, E3 +165949.404}
SPL {X  -160.000, Y  +403.994, Z    +0.000, E1   +31.033, E3 +165968.559}
SPL {X  -160.000, Y  +399.052, Z    +0.000, E1   +31.010, E3 +165986.027}
SPL {X  -160.000, Y  +394.012, Z    +0.000, E1   +31.036, E3 +166003.816}
SPL {X  -159.999, Y  +388.376, Z    +0.000, E1   +31.028, E3 +166023.746}
SPL {X  -159.897, Y  +383.070, Z    +0.000, E1   +31.010, E3 +166042.584}
SPL {X  -159.656, Y  +378.313, Z    +0.000, E1   +30.961, E3 +166059.676}
SPL {X  -159.237, Y  +373.190, Z    +0.000, E1   +30.917, E3 +166078.176}
SPL {X  -158.628, Y  +367.891, Z    +0.000, E1   +30.812, E3 +166097.562}
SPL {X  -157.915, Y  +363.053, Z    +0.000, E1   +30.689, E3 +166115.429}
SPL {X  -157.216, Y  +359.084, Z    +0.000, E1   +30.550, E3 +166130.231}
SPL {X  -156.248, Y  +354.355, Z    +0.000, E1   +30.460, E3 +166147.844}
SPL {X  -155.629, Y  +351.657, Z    +0.000, E1   +25.972, E3 +166194.272}
ENDSPLINE

SPLINE
SPL {X  -156.240, Y  +354.319, Z    +0.000, E1   +23.538, E3 +166206.880}
SPL {X  -159.137, Y  +372.201, Z    +0.000, E1   +12.017, E3 +166236.717}
SPL {X  -159.858, Y  +382.069, Z    +0.000, E1    +5.945, E3 +166243.235}
SPL {X  -160.000, Y  +389.339, Z    +0.000, E1    +1.101, E3 +166246.397}
SPL {X  -160.000, Y  +395.749, Z    +0.000, E1    -3.722, E3 +166249.002}
SPL {X  -160.000, Y  +403.128, Z    +0.000, E1    -9.899, E3 +166252.306}
SPL {X  -160.000, Y  +411.609, Z    +0.000, E1   -16.851, E3 +166257.627}
SPL {X  -160.000, Y  +429.715, Z    +0.000, E1   -27.376, E3 +166276.991}
SPL {X  -160.000, Y  +449.791, Z    +0.000, E1   -32.145, E3 +166318.228}
SPL {X  -160.000, Y  +454.903, Z    +0.000, E1   -32.134, E3 +166335.532}
SPL {X  -160.000, Y  +460.041, Z    +0.000, E1   -32.144, E3 +166352.885}
SPL {X  -160.000, Y  +465.466, Z    +0.000, E1   -32.152, E3 +166371.203}
SPL {X  -160.000, Y  +471.112, Z    +0.000, E1   -32.154, E3 +166390.291}
SPL {X  -160.000, Y  +476.735, Z    +0.000, E1   -32.156, E3 +166409.282}
SPL {X  -160.000, Y  +482.675, Z    +0.000, E1   -32.169, E3 +166429.331}
SPL {X  -160.000, Y  +488.008, Z    +0.000, E1   -32.144, E3 +166447.378}
SPL {X  -160.000, Y  +493.245, Z    +0.000, E1   -32.159, E3 +166465.086}
SPL {X  -160.000, Y  +498.210, Z    +0.000, E1   -32.128, E3 +166481.921}
SPL {X  -160.000, Y  +503.407, Z    +0.000, E1   -32.165, E3 +166499.424}
SPL {X  -160.000, Y  +509.142, Z    +0.000, E1   -32.157, E3 +166518.820}
SPL {X  -160.000, Y  +514.696, Z    +0.000, E1   -32.156, E3 +166537.600}
SPL {X  -160.000, Y  +520.339, Z    +0.000, E1   -32.159, E3 +166556.673}
SPL {X  -160.000, Y  +525.825, Z    +0.000, E1   -32.148, E3 +166575.236}
SPL {X  -160.000, Y  +530.379, Z    +0.000, E1   -32.130, E3 +166590.664}
SPL {X  -160.000, Y  +535.020, Z    +0.000, E1   -32.146, E3 +166606.310}
SPL {X  -160.000, Y  +540.303, Z    +0.000, E1   -32.158, E3 +166624.136}
SPL {X  -160.000, Y  +545.740, Z    +0.000, E1   -32.155, E3 +166642.528}
SPL {X  -160.000, Y  +550.807, Z    +0.000, E1   -32.147, E3 +166659.651}
SPL {X  -160.000, Y  +555.841, Z    +0.000, E1   -32.148, E3 +166676.690}
SPL {X  -160.000, Y  +561.018, Z    +0.000, E1   -32.143, E3 +166694.219}
SPL {X  -160.000, Y  +566.466, Z    +0.000, E1   -32.153, E3 +166712.637}
SPL {X  -160.000, Y  +571.733, Z    +0.000, E1   -32.135, E3 +166730.474}
SPL {X  -160.000, Y  +576.943, Z    +0.000, E1   -32.148, E3 +166748.071}
SPL {X  -160.000, Y  +582.183, Z    +0.000, E1   -32.140, E3 +166765.795}
SPL {X  -160.000, Y  +587.036, Z    +0.000, E1   -32.141, E3 +166782.166}
SPL {X  -160.000, Y  +591.785, Z    +0.000, E1   -32.144, E3 +166798.190}
SPL {X  -160.000, Y  +596.962, Z    +0.000, E1   -32.161, E3 +166815.677}
SPL {X  -160.000, Y  +601.800, Z    +0.000, E1   -32.134, E3 +166832.074}
SPL {X  -160.000, Y  +606.611, Z    +0.000, E1   -32.156, E3 +166848.288}
SPL {X  -160.000, Y  +611.219, Z    +0.000, E1   -32.131, E3 +166863.902}
SPL {X  -160.000, Y  +616.331, Z    +0.000, E1   -32.174, E3 +166881.099}
SPL {X  -160.000, Y  +621.751, Z    +0.000, E1   -32.150, E3 +166899.442}
SPL {X  -160.000, Y  +626.312, Z    +0.000, E1   -32.145, E3 +166914.848}
SPL {X  -160.000, Y  +630.971, Z    +0.000, E1   -32.155, E3 +166930.576}
SPL {X  -160.000, Y  +635.550, Z    +0.000, E1   -32.137, E3 +166946.102}
SPL {X  -160.000, Y  +640.419, Z    +0.000, E1   -32.158, E3 +166962.540}
SPL {X  -160.000, Y  +645.749, Z    +0.000, E1   -32.151, E3 +166980.565}
SPL {X  -160.000, Y  +650.662, Z    +0.000, E1   -32.150, E3 +166997.136}
SPL {X  -160.000, Y  +655.372, Z    +0.000, E1   -32.145, E3 +167013.083}
SPL {X  -160.000, Y  +660.593, Z    +0.000, E1   -32.163, E3 +167030.701}
SPL {X  -160.000, Y  +665.836, Z    +0.000, E1   -32.154, E3 +167048.417}
SPL {X  -160.000, Y  +670.613, Z    +0.000, E1   -32.138, E3 +167064.628}
SPL {X  -159.954, Y  +675.336, Z    +0.000, E1   -32.135, E3 +167080.636}
SPL {X  -159.758, Y  +680.302, Z    +0.000, E1   -32.108, E3 +167097.651}
SPL {X  -159.416, Y  +685.158, Z    +0.000, E1   -32.039, E3 +167114.462}
SPL {X  -158.953, Y  +689.772, Z    +0.000, E1   -31.965, E3 +167130.561}
SPL {X  -158.363, Y  +694.328, Z    +0.000, E1   -31.871, E3 +167146.574}
SPL {X  -157.606, Y  +699.074, Z    +0.000, E1   -31.756, E3 +167163.417}
SPL {X  -156.791, Y  +703.384, Z    +0.000, E1   -31.607, E3 +167178.868}
SPL {X  -155.792, Y  +707.952, Z    +0.000, E1   -31.465, E3 +167195.314}
SPL {X  -155.149, Y  +710.598, Z    +0.000, E1   -26.183, E3 +167250.774}
ENDSPLINE

SPLINE
SPL {X  -158.679, Y  +692.020, Z    +0.000, E1   -14.212, E3 +167284.450}
SPL {X  -159.747, Y  +680.500, Z    +0.000, E1    -7.378, E3 +167292.828}
SPL {X  -160.000, Y  +671.618, Z    +0.000, E1    -1.592, E3 +167296.442}
SPL {X  -160.000, Y  +666.041, Z    +0.000, E1    +2.615, E3 +167298.409}
SPL {X  -160.000, Y  +661.396, Z    +0.000, E1    +6.484, E3 +167300.081}
SPL {X  -160.000, Y  +653.532, Z    +0.000, E1   +13.136, E3 +167304.202}
SPL {X  -160.000, Y  +631.927, Z    +0.000, E1   +26.832, E3 +167326.968}
SPL {X  -160.000, Y  +610.736, Z    +0.000, E1   +32.114, E3 +167369.638}
SPL {X  -160.000, Y  +605.907, Z    +0.000, E1   +32.114, E3 +167385.986}
SPL {X  -160.000, Y  +601.221, Z    +0.000, E1   +32.108, E3 +167401.854}
SPL {X  -160.000, Y  +596.433, Z    +0.000, E1   +32.120, E3 +167418.036}
SPL {X  -160.000, Y  +592.025, Z    +0.000, E1   +32.104, E3 +167432.960}
SPL {X  -160.000, Y  +587.734, Z    +0.000, E1   +32.110, E3 +167447.481}
SPL {X  -160.000, Y  +583.150, Z    +0.000, E1   +32.111, E3 +167463.008}
SPL {X  -160.000, Y  +579.063, Z    +0.000, E1   +32.085, E3 +167476.910}
SPL {X  -160.000, Y  +574.897, Z    +0.000, E1   +32.110, E3 +167490.961}
SPL {X  -160.000, Y  +570.471, Z    +0.000, E1   +32.093, E3 +167505.975}
SPL {X  -160.000, Y  +566.667, Z    +0.000, E1   +32.086, E3 +167518.890}
SPL {X  -160.000, Y  +562.434, Z    +0.000, E1   +32.097, E3 +167533.199}
SPL {X  -160.000, Y  +557.710, Z    +0.000, E1   +32.104, E3 +167549.183}
SPL {X  -160.000, Y  +553.479, Z    +0.000, E1   +32.081, E3 +167563.552}
SPL {X  -160.000, Y  +547.489, Z    +0.000, E1   +32.181, E3 +167583.670}
SPL {X  -160.000, Y  +541.554, Z    +0.000, E1   +32.092, E3 +167603.908}
SPL {X  -160.000, Y  +537.332, Z    +0.000, E1   +32.092, E3 +167618.205}
SPL {X  -160.000, Y  +533.113, Z    +0.000, E1   +32.090, E3 +167632.502}
SPL {X  -160.000, Y  +528.875, Z    +0.000, E1   +32.090, E3 +167646.845}
SPL {X  -160.000, Y  +524.453, Z    +0.000, E1   +32.104, E3 +167661.769}
SPL {X  -160.000, Y  +520.037, Z    +0.000, E1   +32.096, E3 +167676.711}
SPL {X  -160.000, Y  +514.030, Z    +0.000, E1   +32.182, E3 +167696.907}
SPL {X  -160.000, Y  +508.131, Z    +0.000, E1   +32.099, E3 +167717.011}
SPL {X  -160.000, Y  +504.077, Z    +0.000, E1   +32.094, E3 +167730.734}
SPL {X  -160.000, Y  +494.657, Z    +0.000, E1   +34.509, E3 +167745.597}
SPL {X  -160.000, Y  +491.565, Z    +0.000, E1   +33.823, E3 +167759.504}
SPL {X  -160.000, Y  +489.317, Z    +0.000, E1   +32.894, E3 +167772.849}
SPL {X  -160.000, Y  +486.958, Z    +0.000, E1   +31.703, E3 +167788.621}
SPL {X  -160.000, Y  +484.144, Z    +0.000, E1   +30.999, E3 +167803.044}
SPL {X  -160.000, Y  +479.156, Z    +0.000, E1   +31.035, E3 +167820.610}
SPL {X  -160.000, Y  +474.045, Z    +0.000, E1   +31.015, E3 +167838.702}
SPL {X  -160.000, Y  +468.999, Z    +0.000, E1   +31.021, E3 +167856.527}
SPL {X  -160.000, Y  +464.107, Z    +0.000, E1   +31.012, E3 +167873.827}
SPL {X  -160.000, Y  +459.262, Z    +0.000, E1   +31.016, E3 +167890.934}
SPL {X  -160.000, Y  +454.119, Z    +0.000, E1   +31.026, E3 +167909.083}
SPL {X  -160.000, Y  +448.874, Z    +0.000, E1   +31.019, E3 +167927.639}
SPL {X  -160.000, Y  +443.892, Z    +0.000, E1   +31.019, E3 +167945.227}
SPL {X  -160.000, Y  +438.782, Z    +0.000, E1   +31.022, E3 +167963.301}
SPL {X  -160.000, Y  +433.722, Z    +0.000, E1   +31.007, E3 +167981.245}
SPL {X  -160.000, Y  +428.980, Z    +0.000, E1   +31.004, E3 +167998.002}
SPL {X  -160.000, Y  +424.339, Z    +0.000, E1   +31.006, E3 +168014.377}
SPL {X  -160.000, Y  +419.231, Z    +0.000, E1   +31.030, E3 +168032.370}
SPL {X  -160.000, Y  +414.179, Z    +0.000, E1   +31.008, E3 +168050.268}
SPL {X  -160.000, Y  +409.416, Z    +0.000, E1   +31.023, E3 +168067.051}
SPL {X  -160.000, Y  +403.994, Z    +0.000, E1   +31.033, E3 +168086.206}
SPL {X  -160.000, Y  +399.052, Z    +0.000, E1   +31.010, E3 +168103.674}
SPL {X  -160.000, Y  +394.012, Z    +0.000, E1   +31.036, E3 +168121.463}
SPL {X  -159.999, Y  +388.376, Z    +0.000, E1   +31.028, E3 +168141.393}
SPL {X  -159.897, Y  +383.070, Z    +0.000, E1   +31.010, E3 +168160.231}
SPL {X  -159.656, Y  +378.313, Z    +0.000, E1   +30.961, E3 +168177.323}
SPL {X  -159.237, Y  +373.190, Z    +0.000, E1   +30.917, E3 +168195.823}
SPL {X  -158.628, Y  +367.891, Z    +0.000, E1   +30.812, E3 +168215.209}
SPL {X  -157.915, Y  +363.053, Z    +0.000, E1   +30.689, E3 +168233.076}
SPL {X  -157.216, Y  +359.084, Z    +0.000, E1   +30.550, E3 +168247.879}
SPL {X  -156.248, Y  +354.355, Z    +0.000, E1   +30.460, E3 +168265.491}
SPL {X  -155.629, Y  +351.657, Z    +0.000, E1   +25.972, E3 +168311.919}
ENDSPLINE

SPLINE
SPL {X  -156.240, Y  +354.319, Z    +0.000, E1   +23.538, E3 +168324.527}
SPL {X  -159.137, Y  +372.201, Z    +0.000, E1   +12.017, E3 +168354.364}
SPL {X  -159.858, Y  +382.069, Z    +0.000, E1    +5.945, E3 +168360.882}
SPL {X  -160.000, Y  +389.339, Z    +0.000, E1    +1.101, E3 +168364.044}
SPL {X  -160.000, Y  +395.749, Z    +0.000, E1    -3.722, E3 +168366.649}
SPL {X  -160.000, Y  +403.128, Z    +0.000, E1    -9.899, E3 +168369.953}
SPL {X  -160.000, Y  +411.609, Z    +0.000, E1   -16.851, E3 +168375.274}
SPL {X  -160.000, Y  +429.715, Z    +0.000, E1   -27.376, E3 +168394.638}
SPL {X  -160.000, Y  +449.791, Z    +0.000, E1   -32.145, E3 +168435.875}
SPL {X  -160.000, Y  +454.903, Z    +0.000, E1   -32.134, E3 +168453.179}
SPL {X  -160.000, Y  +460.041, Z    +0.000, E1   -32.144, E3 +168470.533}
SPL {X  -160.000, Y  +465.466, Z    +0.000, E1   -32.152, E3 +168488.851}
SPL {X  -160.000, Y  +471.112, Z    +0.000, E1   -32.154, E3 +168507.939}
SPL {X  -160.000, Y  +476.735, Z    +0.000, E1   -32.156, E3 +168526.930}
SPL {X  -160.000, Y  +482.675, Z    +0.000, E1   -32.169, E3 +168546.978}
SPL {X  -160.000, Y  +488.008, Z    +0.000, E1   -32.144, E3 +168565.025}
SPL {X  -160.000, Y  +493.245, Z    +0.000, E1   -32.159, E3 +168582.733}
SPL {X  -160.000, Y  +498.210, Z    +0.000, E1   -32.128, E3 +168599.568}
SPL {X  -160.000, Y  +503.407, Z    +0.000, E1   -32.165, E3 +168617.072}
SPL {X  -160.000, Y  +509.142, Z    +0.000, E1   -32.157, E3 +168636.467}
SPL {X  -160.000, Y  +514.696, Z    +0.000, E1   -32.156, E3 +168655.248}
SPL {X  -160.000, Y  +520.339, Z    +0.000, E1   -32.159, E3 +168674.320}
SPL {X  -160.000, Y  +525.825, Z    +0.000, E1   -32.148, E3 +168692.883}
SPL {X  -160.000, Y  +530.379, Z    +0.000, E1   -32.130, E3 +168708.312}
SPL {X  -160.000, Y  +535.020, Z    +0.000, E1   -32.146, E3 +168723.958}
SPL {X  -160.000, Y  +540.303, Z    +0.000, E1   -32.158, E3 +168741.783}
SPL {X  -160.000, Y  +545.740, Z    +0.000, E1   -32.155, E3 +168760.176}
SPL {X  -160.000, Y  +550.807, Z    +0.000, E1   -32.147, E3 +168777.298}
SPL {X  -160.000, Y  +555.841, Z    +0.000, E1   -32.148, E3 +168794.338}
SPL {X  -160.000, Y  +561.018, Z    +0.000, E1   -32.143, E3 +168811.866}
SPL {X  -160.000, Y  +566.466, Z    +0.000, E1   -32.153, E3 +168830.284}
SPL {X  -160.000, Y  +571.733, Z    +0.000, E1   -32.135, E3 +168848.121}
SPL {X  -160.000, Y  +576.943, Z    +0.000, E1   -32.148, E3 +168865.718}
SPL {X  -160.000, Y  +582.183, Z    +0.000, E1   -32.140, E3 +168883.443}
SPL {X  -160.000, Y  +587.036, Z    +0.000, E1   -32.141, E3 +168899.814}
SPL {X  -160.000, Y  +591.785, Z    +0.000, E1   -32.144, E3 +168915.837}
SPL {X  -160.000, Y  +596.962, Z    +0.000, E1   -32.161, E3 +168933.324}
SPL {X  -160.000, Y  +601.800, Z    +0.000, E1   -32.134, E3 +168949.721}
SPL {X  -160.000, Y  +606.611, Z    +0.000, E1   -32.156, E3 +168965.935}
SPL {X  -160.000, Y  +611.219, Z    +0.000, E1   -32.131, E3 +168981.549}
SPL {X  -160.000, Y  +616.331, Z    +0.000, E1   -32.174, E3 +168998.746}
SPL {X  -160.000, Y  +621.751, Z    +0.000, E1   -32.150, E3 +169017.089}
SPL {X  -160.000, Y  +626.312, Z    +0.000, E1   -32.145, E3 +169032.495}
SPL {X  -160.000, Y  +630.971, Z    +0.000, E1   -32.155, E3 +169048.223}
SPL {X  -160.000, Y  +635.550, Z    +0.000, E1   -32.137, E3 +169063.749}
SPL {X  -160.000, Y  +640.419, Z    +0.000, E1   -32.158, E3 +169080.187}
SPL {X  -160.000, Y  +645.749, Z    +0.000, E1   -32.151, E3 +169098.213}
SPL {X  -160.000, Y  +650.662, Z    +0.000, E1   -32.150, E3 +169114.784}
SPL {X  -160.000, Y  +655.372, Z    +0.000, E1   -32.145, E3 +169130.730}
SPL {X  -160.000, Y  +660.593, Z    +0.000, E1   -32.163, E3 +169148.348}
SPL {X  -160.000, Y  +665.836, Z    +0.000, E1   -32.154, E3 +169166.065}
SPL {X  -160.000, Y  +670.613, Z    +0.000, E1   -32.138, E3 +169182.275}
SPL {X  -159.954, Y  +675.336, Z    +0.000, E1   -32.135, E3 +169198.283}
SPL {X  -159.758, Y  +680.302, Z    +0.000, E1   -32.108, E3 +169215.298}
SPL {X  -159.416, Y  +685.158, Z    +0.000, E1   -32.039, E3 +169232.109}
SPL {X  -158.953, Y  +689.772, Z    +0.000, E1   -31.965, E3 +169248.209}
SPL {X  -158.363, Y  +694.328, Z    +0.000, E1   -31.871, E3 +169264.221}
SPL {X  -157.606, Y  +699.074, Z    +0.000, E1   -31.756, E3 +169281.064}
SPL {X  -156.791, Y  +703.384, Z    +0.000, E1   -31.607, E3 +169296.515}
SPL {X  -155.792, Y  +707.952, Z    +0.000, E1   -31.465, E3 +169312.961}
SPL {X  -155.149, Y  +710.598, Z    +0.000, E1   -26.183, E3 +169368.421}
ENDSPLINE

SPLINE
SPL {X  -158.679, Y  +692.020, Z    +0.000, E1   -14.212, E3 +169402.097}
SPL {X  -159.747, Y  +680.500, Z    +0.000, E1    -7.378, E3 +169410.475}
SPL {X  -160.000, Y  +671.618, Z    +0.000, E1    -1.592, E3 +169414.089}
SPL {X  -160.000, Y  +666.041, Z    +0.000, E1    +2.615, E3 +169416.056}
SPL {X  -160.000, Y  +661.396, Z    +0.000, E1    +6.484, E3 +169417.729}
SPL {X  -160.000, Y  +653.532, Z    +0.000, E1   +13.136, E3 +169421.849}
SPL {X  -160.000, Y  +631.927, Z    +0.000, E1   +26.832, E3 +169444.616}
SPL {X  -160.000, Y  +610.736, Z    +0.000, E1   +32.114, E3 +169487.285}
SPL {X  -160.000, Y  +605.907, Z    +0.000, E1   +32.114, E3 +169503.633}
SPL {X  -160.000, Y  +601.221, Z    +0.000, E1   +32.108, E3 +169519.501}
SPL {X  -160.000, Y  +596.433, Z    +0.000, E1   +32.120, E3 +169535.683}
SPL {X  -160.000, Y  +592.025, Z    +0.000, E1   +32.104, E3 +169550.608}
SPL {X  -160.000, Y  +587.734, Z    +0.000, E1   +32.110, E3 +169565.128}
SPL {X  -160.000, Y  +583.150, Z    +0.000, E1   +32.111, E3 +169580.655}
SPL {X  -160.000, Y  +579.063, Z    +0.000, E1   +32.085, E3 +169594.557}
SPL {X  -160.000, Y  +574.897, Z    +0.000, E1   +32.110, E3 +169608.608}
SPL {X  -160.000, Y  +570.471, Z    +0.000, E1   +32.093, E3 +169623.623}
SPL {X  -160.000, Y  +566.667, Z    +0.000, E1   +32.086, E3 +169636.537}
SPL {X  -160.000, Y  +562.434, Z    +0.000, E1   +32.097, E3 +169650.847}
SPL {X  -160.000, Y  +557.710, Z    +0.000, E1   +32.104, E3 +169666.830}
SPL {X  -160.000, Y  +553.479, Z    +0.000, E1   +32.081, E3 +169681.199}
SPL {X  -160.000, Y  +547.489, Z    +0.000, E1   +32.181, E3 +169701.318}
SPL {X  -160.000, Y  +541.554, Z    +0.000, E1   +32.092, E3 +169721.555}
SPL {X  -160.000, Y  +537.332, Z    +0.000, E1   +32.092, E3 +169735.852}
SPL {X  -160.000, Y  +533.113, Z    +0.000, E1   +32.090, E3 +169750.149}
SPL {X  -160.000, Y  +528.875, Z    +0.000, E1   +32.090, E3 +169764.492}
SPL {X  -160.000, Y  +524.453, Z    +0.000, E1   +32.104, E3 +169779.416}
SPL {X  -160.000, Y  +520.037, Z    +0.000, E1   +32.096, E3 +169794.358}
SPL {X  -160.000, Y  +514.030, Z    +0.000, E1   +32.182, E3 +169814.554}
SPL {X  -160.000, Y  +508.131, Z    +0.000, E1   +32.099, E3 +169834.659}
SPL {X  -160.000, Y  +504.077, Z    +0.000, E1   +32.094, E3 +169848.382}
SPL {X  -160.000, Y  +494.657, Z    +0.000, E1   +34.509, E3 +169863.244}
SPL {X  -160.000, Y  +491.565, Z    +0.000, E1   +33.823, E3 +169877.152}
SPL {X  -160.000, Y  +489.317, Z    +0.000, E1   +32.894, E3 +169890.497}
SPL {X  -160.000, Y  +486.958, Z    +0.000, E1   +31.703, E3 +169906.268}
SPL {X  -160.000, Y  +484.144, Z    +0.000, E1   +30.999, E3 +169920.691}
SPL {X  -160.000, Y  +479.156, Z    +0.000, E1   +31.035, E3 +169938.257}
SPL {X  -160.000, Y  +474.045, Z    +0.000, E1   +31.015, E3 +169956.349}
SPL {X  -160.000, Y  +468.999, Z    +0.000, E1   +31.021, E3 +169974.174}
SPL {X  -160.000, Y  +464.107, Z    +0.000, E1   +31.012, E3 +169991.474}
SPL {X  -160.000, Y  +459.262, Z    +0.000, E1   +31.016, E3 +170008.581}
SPL {X  -160.000, Y  +454.119, Z    +0.000, E1   +31.026, E3 +170026.730}
SPL {X  -160.000, Y  +448.874, Z    +0.000, E1   +31.019, E3 +170045.286}
SPL {X  -160.000, Y  +443.892, Z    +0.000, E1   +31.019, E3 +170062.874}
SPL {X  -160.000, Y  +438.782, Z    +0.000, E1   +31.022, E3 +170080.949}
SPL {X  -160.000, Y  +433.722, Z    +0.000, E1   +31.007, E3 +170098.893}
SPL {X  -160.000, Y  +428.980, Z    +0.000, E1   +31.004, E3 +170115.650}
SPL {X  -160.000, Y  +424.339, Z    +0.000, E1   +31.006, E3 +170132.024}
SPL {X  -160.000, Y  +419.231, Z    +0.000, E1   +31.030, E3 +170150.018}
SPL {X  -160.000, Y  +414.179, Z    +0.000, E1   +31.008, E3 +170167.915}
SPL {X  -160.000, Y  +409.416, Z    +0.000, E1   +31.023, E3 +170184.698}
SPL {X  -160.000, Y  +403.994, Z    +0.000, E1   +31.033, E3 +170203.854}
SPL {X  -160.000, Y  +399.052, Z    +0.000, E1   +31.010, E3 +170221.322}
SPL {X  -160.000, Y  +394.012, Z    +0.000, E1   +31.036, E3 +170239.110}
SPL {X  -159.999, Y  +388.376, Z    +0.000, E1   +31.028, E3 +170259.040}
SPL {X  -159.897, Y  +383.070, Z    +0.000, E1   +31.010, E3 +170277.878}
SPL {X  -159.656, Y  +378.313, Z    +0.000, E1   +30.961, E3 +170294.970}
SPL {X  -159.237, Y  +373.190, Z    +0.000, E1   +30.917, E3 +170313.471}
SPL {X  -158.628, Y  +367.891, Z    +0.000, E1   +30.812, E3 +170332.856}
SPL {X  -157.915, Y  +363.053, Z    +0.000, E1   +30.689, E3 +170350.723}
SPL {X  -157.216, Y  +359.084, Z    +0.000, E1   +30.550, E3 +170365.526}
SPL {X  -156.248, Y  +354.355, Z    +0.000, E1   +30.460, E3 +170383.138}
SPL {X  -155.629, Y  +351.657, Z    +0.000, E1   +25.972, E3 +170429.567}
ENDSPLINE

SPLINE
SPL {X  -156.240, Y  +354.319, Z    +0.000, E1   +23.538, E3 +170442.174}
SPL {X  -159.137, Y  +372.201, Z    +0.000, E1   +12.017, E3 +170472.011}
SPL {X  -159.858, Y  +382.069, Z    +0.000, E1    +5.945, E3 +170478.529}
SPL {X  -160.000, Y  +389.339, Z    +0.000, E1    +1.101, E3 +170481.691}
SPL {X  -160.000, Y  +395.749, Z    +0.000, E1    -3.722, E3 +170484.297}
SPL {X  -160.000, Y  +403.128, Z    +0.000, E1    -9.899, E3 +170487.601}
SPL {X  -160.000, Y  +411.609, Z    +0.000, E1   -16.851, E3 +170492.922}
SPL {X  -160.000, Y  +429.715, Z    +0.000, E1   -27.376, E3 +170512.285}
SPL {X  -160.000, Y  +449.791, Z    +0.000, E1   -32.145, E3 +170553.522}
SPL {X  -160.000, Y  +454.903, Z    +0.000, E1   -32.134, E3 +170570.827}
SPL {X  -160.000, Y  +460.041, Z    +0.000, E1   -32.144, E3 +170588.180}
SPL {X  -160.000, Y  +465.466, Z    +0.000, E1   -32.152, E3 +170606.498}
SPL {X  -160.000, Y  +471.112, Z    +0.000, E1   -32.154, E3 +170625.586}
SPL {X  -160.000, Y  +476.735, Z    +0.000, E1   -32.156, E3 +170644.577}
SPL {X  -160.000, Y  +482.675, Z    +0.000, E1   -32.169, E3 +170664.626}
SPL {X  -160.000, Y  +488.008, Z    +0.000, E1   -32.144, E3 +170682.672}
SPL {X  -160.000, Y  +493.245, Z    +0.000, E1   -32.159, E3 +170700.380}
SPL {X  -160.000, Y  +498.210, Z    +0.000, E1   -32.128, E3 +170717.215}
SPL {X  -160.000, Y  +503.407, Z    +0.000, E1   -32.165, E3 +170734.719}
SPL {X  -160.000, Y  +509.142, Z    +0.000, E1   -32.157, E3 +170754.114}
SPL {X  -160.000, Y  +514.696, Z    +0.000, E1   -32.156, E3 +170772.895}
SPL {X  -160.000, Y  +520.339, Z    +0.000, E1   -32.159, E3 +170791.967}
SPL {X  -160.000, Y  +525.825, Z    +0.000, E1   -32.148, E3 +170810.531}
SPL {X  -160.000, Y  +530.379, Z    +0.000, E1   -32.130, E3 +170825.959}
SPL {X  -160.000, Y  +535.020, Z    +0.000, E1   -32.146, E3 +170841.605}
SPL {X  -160.000, Y  +540.303, Z    +0.000, E1   -32.158, E3 +170859.430}
SPL {X  -160.000, Y  +545.740, Z    +0.000, E1   -32.155, E3 +170877.823}
SPL {X  -160.000, Y  +550.807, Z    +0.000, E1   -32.147, E3 +170894.945}
SPL {X  -160.000, Y  +555.841, Z    +0.000, E1   -32.148, E3 +170911.985}
SPL {X  -160.000, Y  +561.018, Z    +0.000, E1   -32.143, E3 +170929.514}
SPL {X  -160.000, Y  +566.466, Z    +0.000, E1   -32.153, E3 +170947.932}
SPL {X  -160.000, Y  +571.733, Z    +0.000, E1   -32.135, E3 +170965.768}
SPL {X  -160.000, Y  +576.943, Z    +0.000, E1   -32.148, E3 +170983.365}
SPL {X  -160.000, Y  +582.183, Z    +0.000, E1   -32.140, E3 +171001.090}
SPL {X  -160.000, Y  +587.036, Z    +0.000, E1   -32.141, E3 +171017.461}
SPL {X  -160.000, Y  +591.785, Z    +0.000, E1   -32.144, E3 +171033.485}
SPL {X  -160.000, Y  +596.962, Z    +0.000, E1   -32.161, E3 +171050.971}
SPL {X  -160.000, Y  +601.800, Z    +0.000, E1   -32.134, E3 +171067.368}
SPL {X  -160.000, Y  +606.611, Z    +0.000, E1   -32.156, E3 +171083.583}
SPL {X  -160.000, Y  +611.219, Z    +0.000, E1   -32.131, E3 +171099.196}
SPL {X  -160.000, Y  +616.331, Z    +0.000, E1   -32.174, E3 +171116.394}
SPL {X  -160.000, Y  +621.751, Z    +0.000, E1   -32.150, E3 +171134.736}
SPL {X  -160.000, Y  +626.312, Z    +0.000, E1   -32.145, E3 +171150.142}
SPL {X  -160.000, Y  +630.971, Z    +0.000, E1   -32.155, E3 +171165.870}
SPL {X  -160.000, Y  +635.550, Z    +0.000, E1   -32.137, E3 +171181.396}
SPL {X  -160.000, Y  +640.419, Z    +0.000, E1   -32.158, E3 +171197.834}
SPL {X  -160.000, Y  +645.749, Z    +0.000, E1   -32.151, E3 +171215.860}
SPL {X  -160.000, Y  +650.662, Z    +0.000, E1   -32.150, E3 +171232.431}
SPL {X  -160.000, Y  +655.372, Z    +0.000, E1   -32.145, E3 +171248.378}
SPL {X  -160.000, Y  +660.593, Z    +0.000, E1   -32.163, E3 +171265.995}
SPL {X  -160.000, Y  +665.836, Z    +0.000, E1   -32.154, E3 +171283.712}
SPL {X  -160.000, Y  +670.613, Z    +0.000, E1   -32.138, E3 +171299.922}
SPL {X  -159.954, Y  +675.336, Z    +0.000, E1   -32.135, E3 +171315.931}
SPL {X  -159.758, Y  +680.302, Z    +0.000, E1   -32.108, E3 +171332.945}
SPL {X  -159.416, Y  +685.158, Z    +0.000, E1   -32.039, E3 +171349.757}
SPL {X  -158.953, Y  +689.772, Z    +0.000, E1   -31.965, E3 +171365.856}
SPL {X  -158.363, Y  +694.328, Z    +0.000, E1   -31.871, E3 +171381.869}
SPL {X  -157.606, Y  +699.074, Z    +0.000, E1   -31.756, E3 +171398.712}
SPL {X  -156.791, Y  +703.384, Z    +0.000, E1   -31.607, E3 +171414.162}
SPL {X  -155.792, Y  +707.952, Z    +0.000, E1   -31.465, E3 +171430.608}
SPL {X  -155.149, Y  +710.598, Z    +0.000, E1   -26.183, E3 +171486.068}
ENDSPLINE

SPLINE
SPL {X  -158.679, Y  +692.020, Z    +0.000, E1   -14.212, E3 +171519.744}
SPL {X  -159.747, Y  +680.500, Z    +0.000, E1    -7.378, E3 +171528.122}
SPL {X  -160.000, Y  +671.618, Z    +0.000, E1    -1.592, E3 +171531.737}
SPL {X  -160.000, Y  +666.041, Z    +0.000, E1    +2.615, E3 +171533.703}
SPL {X  -160.000, Y  +661.396, Z    +0.000, E1    +6.484, E3 +171535.376}
SPL {X  -160.000, Y  +653.532, Z    +0.000, E1   +13.136, E3 +171539.496}
SPL {X  -160.000, Y  +631.927, Z    +0.000, E1   +26.832, E3 +171562.263}
SPL {X  -160.000, Y  +610.736, Z    +0.000, E1   +32.114, E3 +171604.932}
SPL {X  -160.000, Y  +605.907, Z    +0.000, E1   +32.114, E3 +171621.281}
SPL {X  -160.000, Y  +601.221, Z    +0.000, E1   +32.108, E3 +171637.148}
SPL {X  -160.000, Y  +596.433, Z    +0.000, E1   +32.120, E3 +171653.330}
SPL {X  -160.000, Y  +592.025, Z    +0.000, E1   +32.104, E3 +171668.255}
SPL {X  -160.000, Y  +587.734, Z    +0.000, E1   +32.110, E3 +171682.775}
SPL {X  -160.000, Y  +583.150, Z    +0.000, E1   +32.111, E3 +171698.303}
SPL {X  -160.000, Y  +579.063, Z    +0.000, E1   +32.085, E3 +171712.204}
SPL {X  -160.000, Y  +574.897, Z    +0.000, E1   +32.110, E3 +171726.255}
SPL {X  -160.000, Y  +570.471, Z    +0.000, E1   +32.093, E3 +171741.270}
SPL {X  -160.000, Y  +566.667, Z    +0.000, E1   +32.086, E3 +171754.184}
SPL {X  -160.000, Y  +562.434, Z    +0.000, E1   +32.097, E3 +171768.494}
SPL {X  -160.000, Y  +557.710, Z    +0.000, E1   +32.104, E3 +171784.477}
SPL {X  -160.000, Y  +553.479, Z    +0.000, E1   +32.081, E3 +171798.846}
SPL {X  -160.000, Y  +547.489, Z    +0.000, E1   +32.181, E3 +171818.965}
SPL {X  -160.000, Y  +541.554, Z    +0.000, E1   +32.092, E3 +171839.202}
SPL {X  -160.000, Y  +537.332, Z    +0.000, E1   +32.092, E3 +171853.499}
SPL {X  -160.000, Y  +533.113, Z    +0.000, E1   +32.090, E3 +171867.796}
SPL {X  -160.000, Y  +528.875, Z    +0.000, E1   +32.090, E3 +171882.139}
SPL {X  -160.000, Y  +524.453, Z    +0.000, E1   +32.104, E3 +171897.063}
SPL {X  -160.000, Y  +520.037, Z    +0.000, E1   +32.096, E3 +171912.005}
SPL {X  -160.000, Y  +514.030, Z    +0.000, E1   +32.182, E3 +171932.201}
SPL {X  -160.000, Y  +508.131, Z    +0.000, E1   +32.099, E3 +171952.306}
SPL {X  -160.000, Y  +504.077, Z    +0.000, E1   +32.094, E3 +171966.029}
SPL {X  -160.000, Y  +494.657, Z    +0.000, E1   +34.509, E3 +171980.892}
SPL {X  -160.000, Y  +491.565, Z    +0.000, E1   +33.823, E3 +171994.799}
SPL {X  -160.000, Y  +489.317, Z    +0.000, E1   +32.894, E3 +172008.144}
SPL {X  -160.000, Y  +486.958, Z    +0.000, E1   +31.703, E3 +172023.916}
SPL {X  -160.000, Y  +484.144, Z    +0.000, E1   +30.999, E3 +172038.338}
SPL {X  -160.000, Y  +479.156, Z    +0.000, E1   +31.035, E3 +172055.904}
SPL {X  -160.000, Y  +474.045, Z    +0.000, E1   +31.015, E3 +172073.996}
SPL {X  -160.000, Y  +468.999, Z    +0.000, E1   +31.021, E3 +172091.821}
SPL {X  -160.000, Y  +464.107, Z    +0.000, E1   +31.012, E3 +172109.121}
SPL {X  -160.000, Y  +459.262, Z    +0.000, E1   +31.016, E3 +172126.228}
SPL {X  -160.000, Y  +454.119, Z    +0.000, E1   +31.026, E3 +172144.378}
SPL {X  -160.000, Y  +448.874, Z    +0.000, E1   +31.019, E3 +172162.934}
SPL {X  -160.000, Y  +443.892, Z    +0.000, E1   +31.019, E3 +172180.522}
SPL {X  -160.000, Y  +438.782, Z    +0.000, E1   +31.022, E3 +172198.596}
SPL {X  -160.000, Y  +433.722, Z    +0.000, E1   +31.007, E3 +172216.540}
SPL {X  -160.000, Y  +428.980, Z    +0.000, E1   +31.004, E3 +172233.297}
SPL {X  -160.000, Y  +424.339, Z    +0.000, E1   +31.006, E3 +172249.671}
SPL {X  -160.000, Y  +419.231, Z    +0.000, E1   +31.030, E3 +172267.665}
SPL {X  -160.000, Y  +414.179, Z    +0.000, E1   +31.008, E3 +172285.562}
SPL {X  -160.000, Y  +409.416, Z    +0.000, E1   +31.023, E3 +172302.345}
SPL {X  -160.000, Y  +403.994, Z    +0.000, E1   +31.033, E3 +172321.501}
SPL {X  -160.000, Y  +399.052, Z    +0.000, E1   +31.010, E3 +172338.969}
SPL {X  -160.000, Y  +394.012, Z    +0.000, E1   +31.036, E3 +172356.758}
SPL {X  -159.999, Y  +388.376, Z    +0.000, E1   +31.028, E3 +172376.687}
SPL {X  -159.897, Y  +383.070, Z    +0.000, E1   +31.010, E3 +172395.525}
SPL {X  -159.656, Y  +378.313, Z    +0.000, E1   +30.961, E3 +172412.618}
SPL {X  -159.237, Y  +373.190, Z    +0.000, E1   +30.917, E3 +172431.118}
SPL {X  -158.628, Y  +367.891, Z    +0.000, E1   +30.812, E3 +172450.504}
SPL {X  -157.915, Y  +363.053, Z    +0.000, E1   +30.689, E3 +172468.371}
SPL {X  -157.216, Y  +359.084, Z    +0.000, E1   +30.550, E3 +172483.173}
SPL {X  -156.248, Y  +354.355, Z    +0.000, E1   +30.460, E3 +172500.785}
SPL {X  -155.629, Y  +351.657, Z    +0.000, E1   +25.972, E3 +172547.214}
ENDSPLINE

SPLINE
SPL {X  -156.240, Y  +354.319, Z    +0.000, E1   +23.538, E3 +172559.821}
SPL {X  -159.137, Y  +372.201, Z    +0.000, E1   +12.017, E3 +172589.659}
SPL {X  -159.858, Y  +382.069, Z    +0.000, E1    +5.945, E3 +172596.176}
SPL {X  -160.000, Y  +389.339, Z    +0.000, E1    +1.101, E3 +172599.339}
SPL {X  -160.000, Y  +395.749, Z    +0.000, E1    -3.722, E3 +172601.944}
SPL {X  -160.000, Y  +403.128, Z    +0.000, E1    -9.899, E3 +172605.248}
SPL {X  -160.000, Y  +411.609, Z    +0.000, E1   -16.851, E3 +172610.569}
SPL {X  -160.000, Y  +429.715, Z    +0.000, E1   -27.376, E3 +172629.933}
SPL {X  -160.000, Y  +449.791, Z    +0.000, E1   -32.145, E3 +172671.170}
SPL {X  -160.000, Y  +454.903, Z    +0.000, E1   -32.134, E3 +172688.474}
SPL {X  -160.000, Y  +460.041, Z    +0.000, E1   -32.144, E3 +172705.827}
SPL {X  -160.000, Y  +465.466, Z    +0.000, E1   -32.152, E3 +172724.145}
SPL {X  -160.000, Y  +471.112, Z    +0.000, E1   -32.154, E3 +172743.233}
SPL {X  -160.000, Y  +476.735, Z    +0.000, E1   -32.156, E3 +172762.224}
SPL {X  -160.000, Y  +482.675, Z    +0.000, E1   -32.169, E3 +172782.273}
SPL {X  -160.000, Y  +488.008, Z    +0.000, E1   -32.144, E3 +172800.319}
SPL {X  -160.000, Y  +493.245, Z    +0.000, E1   -32.159, E3 +172818.028}
SPL {X  -160.000, Y  +498.210, Z    +0.000, E1   -32.128, E3 +172834.862}
SPL {X  -160.000, Y  +503.407, Z    +0.000, E1   -32.165, E3 +172852.366}
SPL {X  -160.000, Y  +509.142, Z    +0.000, E1   -32.157, E3 +172871.762}
SPL {X  -160.000, Y  +514.696, Z    +0.000, E1   -32.156, E3 +172890.542}
SPL {X  -160.000, Y  +520.339, Z    +0.000, E1   -32.159, E3 +172909.614}
SPL {X  -160.000, Y  +525.825, Z    +0.000, E1   -32.148, E3 +172928.178}
SPL {X  -160.000, Y  +530.379, Z    +0.000, E1   -32.130, E3 +172943.606}
SPL {X  -160.000, Y  +535.020, Z    +0.000, E1   -32.146, E3 +172959.252}
SPL {X  -160.000, Y  +540.303, Z    +0.000, E1   -32.158, E3 +172977.077}
SPL {X  -160.000, Y  +545.740, Z    +0.000, E1   -32.155, E3 +172995.470}
SPL {X  -160.000, Y  +550.807, Z    +0.000, E1   -32.147, E3 +173012.593}
SPL {X  -160.000, Y  +555.841, Z    +0.000, E1   -32.148, E3 +173029.632}
SPL {X  -160.000, Y  +561.018, Z    +0.000, E1   -32.143, E3 +173047.161}
SPL {X  -160.000, Y  +566.466, Z    +0.000, E1   -32.153, E3 +173065.579}
SPL {X  -160.000, Y  +571.733, Z    +0.000, E1   -32.135, E3 +173083.416}
SPL {X  -160.000, Y  +576.943, Z    +0.000, E1   -32.148, E3 +173101.013}
SPL {X  -160.000, Y  +582.183, Z    +0.000, E1   -32.140, E3 +173118.737}
SPL {X  -160.000, Y  +587.036, Z    +0.000, E1   -32.141, E3 +173135.108}
SPL {X  -160.000, Y  +591.785, Z    +0.000, E1   -32.144, E3 +173151.132}
SPL {X  -160.000, Y  +596.962, Z    +0.000, E1   -32.161, E3 +173168.618}
SPL {X  -160.000, Y  +601.800, Z    +0.000, E1   -32.134, E3 +173185.016}
SPL {X  -160.000, Y  +606.611, Z    +0.000, E1   -32.156, E3 +173201.230}
SPL {X  -160.000, Y  +611.219, Z    +0.000, E1   -32.131, E3 +173216.843}
SPL {X  -160.000, Y  +616.331, Z    +0.000, E1   -32.174, E3 +173234.041}
SPL {X  -160.000, Y  +621.751, Z    +0.000, E1   -32.150, E3 +173252.384}
SPL {X  -160.000, Y  +626.312, Z    +0.000, E1   -32.145, E3 +173267.790}
SPL {X  -160.000, Y  +630.971, Z    +0.000, E1   -32.155, E3 +173283.518}
SPL {X  -160.000, Y  +635.550, Z    +0.000, E1   -32.137, E3 +173299.044}
SPL {X  -160.000, Y  +640.419, Z    +0.000, E1   -32.158, E3 +173315.482}
SPL {X  -160.000, Y  +645.749, Z    +0.000, E1   -32.151, E3 +173333.507}
SPL {X  -160.000, Y  +650.662, Z    +0.000, E1   -32.150, E3 +173350.078}
SPL {X  -160.000, Y  +655.372, Z    +0.000, E1   -32.145, E3 +173366.025}
SPL {X  -160.000, Y  +660.593, Z    +0.000, E1   -32.163, E3 +173383.643}
SPL {X  -160.000, Y  +665.836, Z    +0.000, E1   -32.154, E3 +173401.359}
SPL {X  -160.000, Y  +670.613, Z    +0.000, E1   -32.138, E3 +173417.570}
SPL {X  -159.954, Y  +675.336, Z    +0.000, E1   -32.135, E3 +173433.578}
SPL {X  -159.758, Y  +680.302, Z    +0.000, E1   -32.108, E3 +173450.593}
SPL {X  -159.416, Y  +685.158, Z    +0.000, E1   -32.039, E3 +173467.404}
SPL {X  -158.953, Y  +689.772, Z    +0.000, E1   -31.965, E3 +173483.503}
SPL {X  -158.363, Y  +694.328, Z    +0.000, E1   -31.871, E3 +173499.516}
SPL {X  -157.606, Y  +699.074, Z    +0.000, E1   -31.756, E3 +173516.359}
SPL {X  -156.791, Y  +703.384, Z    +0.000, E1   -31.607, E3 +173531.809}
SPL {X  -155.792, Y  +707.952, Z    +0.000, E1   -31.465, E3 +173548.256}
SPL {X  -155.149, Y  +710.598, Z    +0.000, E1   -26.183, E3 +173603.716}
ENDSPLINE

SPLINE
SPL {X  -158.679, Y  +692.020, Z    +0.000, E1   -14.212, E3 +173637.392}
SPL {X  -159.747, Y  +680.500, Z    +0.000, E1    -7.378, E3 +173645.769}
SPL {X  -160.000, Y  +671.618, Z    +0.000, E1    -1.592, E3 +173649.384}
SPL {X  -160.000, Y  +666.041, Z    +0.000, E1    +2.615, E3 +173651.350}
SPL {X  -160.000, Y  +661.396, Z    +0.000, E1    +6.484, E3 +173653.023}
SPL {X  -160.000, Y  +653.532, Z    +0.000, E1   +13.136, E3 +173657.144}
SPL {X  -160.000, Y  +631.927, Z    +0.000, E1   +26.832, E3 +173679.910}
SPL {X  -160.000, Y  +610.736, Z    +0.000, E1   +32.114, E3 +173722.580}
SPL {X  -160.000, Y  +605.907, Z    +0.000, E1   +32.114, E3 +173738.928}
SPL {X  -160.000, Y  +601.221, Z    +0.000, E1   +32.108, E3 +173754.795}
SPL {X  -160.000, Y  +596.433, Z    +0.000, E1   +32.120, E3 +173770.978}
SPL {X  -160.000, Y  +592.025, Z    +0.000, E1   +32.104, E3 +173785.902}
SPL {X  -160.000, Y  +587.734, Z    +0.000, E1   +32.110, E3 +173800.423}
SPL {X  -160.000, Y  +583.150, Z    +0.000, E1   +32.111, E3 +173815.950}
SPL {X  -160.000, Y  +579.063, Z    +0.000, E1   +32.085, E3 +173829.851}
SPL {X  -160.000, Y  +574.897, Z    +0.000, E1   +32.110, E3 +173843.903}
SPL {X  -160.000, Y  +570.471, Z    +0.000, E1   +32.093, E3 +173858.917}
SPL {X  -160.000, Y  +566.667, Z    +0.000, E1   +32.086, E3 +173871.832}
SPL {X  -160.000, Y  +562.434, Z    +0.000, E1   +32.097, E3 +173886.141}
SPL {X  -160.000, Y  +557.710, Z    +0.000, E1   +32.104, E3 +173902.125}
SPL {X  -160.000, Y  +553.479, Z    +0.000, E1   +32.081, E3 +173916.494}
SPL {X  -160.000, Y  +547.489, Z    +0.000, E1   +32.181, E3 +173936.612}
SPL {X  -160.000, Y  +541.554, Z    +0.000, E1   +32.092, E3 +173956.849}
SPL {X  -160.000, Y  +537.332, Z    +0.000, E1   +32.092, E3 +173971.147}
SPL {X  -160.000, Y  +533.113, Z    +0.000, E1   +32.090, E3 +173985.443}
SPL {X  -160.000, Y  +528.875, Z    +0.000, E1   +32.090, E3 +173999.787}
SPL {X  -160.000, Y  +524.453, Z    +0.000, E1   +32.104, E3 +174014.711}
SPL {X  -160.000, Y  +520.037, Z    +0.000, E1   +32.096, E3 +174029.653}
SPL {X  -160.000, Y  +514.030, Z    +0.000, E1   +32.182, E3 +174049.849}
SPL {X  -160.000, Y  +508.131, Z    +0.000, E1   +32.099, E3 +174069.953}
SPL {X  -160.000, Y  +504.077, Z    +0.000, E1   +32.094, E3 +174083.676}
SPL {X  -160.000, Y  +494.657, Z    +0.000, E1   +34.509, E3 +174098.539}
SPL {X  -160.000, Y  +491.565, Z    +0.000, E1   +33.823, E3 +174112.446}
SPL {X  -160.000, Y  +489.317, Z    +0.000, E1   +32.894, E3 +174125.791}
SPL {X  -160.000, Y  +486.958, Z    +0.000, E1   +31.703, E3 +174141.563}
SPL {X  -160.000, Y  +484.144, Z    +0.000, E1   +30.999, E3 +174155.986}
SPL {X  -160.000, Y  +479.156, Z    +0.000, E1   +31.035, E3 +174173.552}
SPL {X  -160.000, Y  +474.045, Z    +0.000, E1   +31.015, E3 +174191.643}
SPL {X  -160.000, Y  +468.999, Z    +0.000, E1   +31.021, E3 +174209.469}
SPL {X  -160.000, Y  +464.107, Z    +0.000, E1   +31.012, E3 +174226.769}
SPL {X  -160.000, Y  +459.262, Z    +0.000, E1   +31.016, E3 +174243.876}
SPL {X  -160.000, Y  +454.119, Z    +0.000, E1   +31.026, E3 +174262.025}
SPL {X  -160.000, Y  +448.874, Z    +0.000, E1   +31.019, E3 +174280.581}
SPL {X  -160.000, Y  +443.892, Z    +0.000, E1   +31.019, E3 +174298.169}
SPL {X  -160.000, Y  +438.782, Z    +0.000, E1   +31.022, E3 +174316.243}
SPL {X  -160.000, Y  +433.722, Z    +0.000, E1   +31.007, E3 +174334.187}
SPL {X  -160.000, Y  +428.980, Z    +0.000, E1   +31.004, E3 +174350.944}
SPL {X  -160.000, Y  +424.339, Z    +0.000, E1   +31.006, E3 +174367.319}
SPL {X  -160.000, Y  +419.231, Z    +0.000, E1   +31.030, E3 +174385.312}
SPL {X  -160.000, Y  +414.179, Z    +0.000, E1   +31.008, E3 +174403.209}
SPL {X  -160.000, Y  +409.416, Z    +0.000, E1   +31.023, E3 +174419.993}
SPL {X  -160.000, Y  +403.994, Z    +0.000, E1   +31.033, E3 +174439.148}
SPL {X  -160.000, Y  +399.052, Z    +0.000, E1   +31.010, E3 +174456.616}
SPL {X  -160.000, Y  +394.012, Z    +0.000, E1   +31.036, E3 +174474.405}
SPL {X  -159.999, Y  +388.376, Z    +0.000, E1   +31.028, E3 +174494.335}
SPL {X  -159.897, Y  +383.070, Z    +0.000, E1   +31.010, E3 +174513.173}
SPL {X  -159.656, Y  +378.313, Z    +0.000, E1   +30.961, E3 +174530.265}
SPL {X  -159.237, Y  +373.190, Z    +0.000, E1   +30.917, E3 +174548.765}
SPL {X  -158.628, Y  +367.891, Z    +0.000, E1   +30.812, E3 +174568.151}
SPL {X  -157.915, Y  +363.053, Z    +0.000, E1   +30.689, E3 +174586.018}
SPL {X  -157.216, Y  +359.084, Z    +0.000, E1   +30.550, E3 +174600.820}
SPL {X  -156.248, Y  +354.355, Z    +0.000, E1   +30.460, E3 +174618.433}
SPL {X  -155.629, Y  +351.657, Z    +0.000, E1   +25.972, E3 +174664.861}
ENDSPLINE

SPLINE
SPL {X  -156.240, Y  +354.319, Z    +0.000, E1   +23.538, E3 +174677.469}
SPL {X  -159.137, Y  +372.201, Z    +0.000, E1   +12.017, E3 +174707.306}
SPL {X  -159.858, Y  +382.069, Z    +0.000, E1    +5.945, E3 +174713.824}
SPL {X  -160.000, Y  +389.339, Z    +0.000, E1    +1.101, E3 +174716.986}
SPL {X  -160.000, Y  +395.749, Z    +0.000, E1    -3.722, E3 +174719.591}
SPL {X  -160.000, Y  +403.128, Z    +0.000, E1    -9.899, E3 +174722.895}
SPL {X  -160.000, Y  +411.609, Z    +0.000, E1   -16.851, E3 +174728.216}
SPL {X  -160.000, Y  +429.715, Z    +0.000, E1   -27.376, E3 +174747.580}
SPL {X  -160.000, Y  +449.791, Z    +0.000, E1   -32.145, E3 +174788.817}
SPL {X  -160.000, Y  +454.903, Z    +0.000, E1   -32.134, E3 +174806.121}
SPL {X  -160.000, Y  +460.041, Z    +0.000, E1   -32.144, E3 +174823.475}
SPL {X  -160.000, Y  +465.466, Z    +0.000, E1   -32.152, E3 +174841.792}
SPL {X  -160.000, Y  +471.112, Z    +0.000, E1   -32.154, E3 +174860.881}
SPL {X  -160.000, Y  +476.735, Z    +0.000, E1   -32.156, E3 +174879.872}
SPL {X  -160.000, Y  +482.675, Z    +0.000, E1   -32.169, E3 +174899.920}
SPL {X  -160.000, Y  +488.008, Z    +0.000, E1   -32.144, E3 +174917.967}
SPL {X  -160.000, Y  +493.245, Z    +0.000, E1   -32.159, E3 +174935.675}
SPL {X  -160.000, Y  +498.210, Z    +0.000, E1   -32.128, E3 +174952.510}
SPL {X  -160.000, Y  +503.407, Z    +0.000, E1   -32.165, E3 +174970.013}
SPL {X  -160.000, Y  +509.142, Z    +0.000, E1   -32.157, E3 +174989.409}
SPL {X  -160.000, Y  +514.696, Z    +0.000, E1   -32.156, E3 +175008.190}
SPL {X  -160.000, Y  +520.339, Z    +0.000, E1   -32.159, E3 +175027.262}
SPL {X  -160.000, Y  +525.825, Z    +0.000, E1   -32.148, E3 +175045.825}
SPL {X  -160.000, Y  +530.379, Z    +0.000, E1   -32.130, E3 +175061.253}
SPL {X  -160.000, Y  +535.020, Z    +0.000, E1   -32.146, E3 +175076.899}
SPL {X  -160.000, Y  +540.303, Z    +0.000, E1   -32.158, E3 +175094.725}
SPL {X  -160.000, Y  +545.740, Z    +0.000, E1   -32.155, E3 +175113.117}
SPL {X  -160.000, Y  +550.807, Z    +0.000, E1   -32.147, E3 +175130.240}
SPL {X  -160.000, Y  +555.841, Z    +0.000, E1   -32.148, E3 +175147.279}
SPL {X  -160.000, Y  +561.018, Z    +0.000, E1   -32.143, E3 +175164.808}
SPL {X  -160.000, Y  +566.466, Z    +0.000, E1   -32.153, E3 +175183.226}
SPL {X  -160.000, Y  +571.733, Z    +0.000, E1   -32.135, E3 +175201.063}
SPL {X  -160.000, Y  +576.943, Z    +0.000, E1   -32.148, E3 +175218.660}
SPL {X  -160.000, Y  +582.183, Z    +0.000, E1   -32.140, E3 +175236.385}
SPL {X  -160.000, Y  +587.036, Z    +0.000, E1   -32.141, E3 +175252.755}
SPL {X  -160.000, Y  +591.785, Z    +0.000, E1   -32.144, E3 +175268.779}
SPL {X  -160.000, Y  +596.962, Z    +0.000, E1   -32.161, E3 +175286.266}
SPL {X  -160.000, Y  +601.800, Z    +0.000, E1   -32.134, E3 +175302.663}
SPL {X  -160.000, Y  +606.611, Z    +0.000, E1   -32.156, E3 +175318.877}
SPL {X  -160.000, Y  +611.219, Z    +0.000, E1   -32.131, E3 +175334.491}
SPL {X  -160.000, Y  +616.331, Z    +0.000, E1   -32.174, E3 +175351.688}
SPL {X  -160.000, Y  +621.751, Z    +0.000, E1   -32.150, E3 +175370.031}
SPL {X  -160.000, Y  +626.312, Z    +0.000, E1   -32.145, E3 +175385.437}
SPL {X  -160.000, Y  +630.971, Z    +0.000, E1   -32.155, E3 +175401.165}
SPL {X  -160.000, Y  +635.550, Z    +0.000, E1   -32.137, E3 +175416.691}
SPL {X  -160.000, Y  +640.419, Z    +0.000, E1   -32.158, E3 +175433.129}
SPL {X  -160.000, Y  +645.749, Z    +0.000, E1   -32.151, E3 +175451.154}
SPL {X  -160.000, Y  +650.662, Z    +0.000, E1   -32.150, E3 +175467.725}
SPL {X  -160.000, Y  +655.372, Z    +0.000, E1   -32.145, E3 +175483.672}
SPL {X  -160.000, Y  +660.593, Z    +0.000, E1   -32.163, E3 +175501.290}
SPL {X  -160.000, Y  +665.836, Z    +0.000, E1   -32.154, E3 +175519.007}
SPL {X  -160.000, Y  +670.613, Z    +0.000, E1   -32.138, E3 +175535.217}
SPL {X  -159.954, Y  +675.336, Z    +0.000, E1   -32.135, E3 +175551.225}
SPL {X  -159.758, Y  +680.302, Z    +0.000, E1   -32.108, E3 +175568.240}
SPL {X  -159.416, Y  +685.158, Z    +0.000, E1   -32.039, E3 +175585.051}
SPL {X  -158.953, Y  +689.772, Z    +0.000, E1   -31.965, E3 +175601.151}
SPL {X  -158.363, Y  +694.328, Z    +0.000, E1   -31.871, E3 +175617.163}
SPL {X  -157.606, Y  +699.074, Z    +0.000, E1   -31.756, E3 +175634.006}
SPL {X  -156.791, Y  +703.384, Z    +0.000, E1   -31.607, E3 +175649.457}
SPL {X  -155.792, Y  +707.952, Z    +0.000, E1   -31.465, E3 +175665.903}
SPL {X  -155.149, Y  +710.598, Z    +0.000, E1   -26.183, E3 +175721.363}
ENDSPLINE

SPLINE
SPL {X  -158.679, Y  +692.020, Z    +0.000, E1   -14.212, E3 +175755.039}
SPL {X  -159.747, Y  +680.500, Z    +0.000, E1    -7.378, E3 +175763.417}
SPL {X  -160.000, Y  +671.618, Z    +0.000, E1    -1.592, E3 +175767.031}
SPL {X  -160.000, Y  +666.041, Z    +0.000, E1    +2.615, E3 +175768.998}
SPL {X  -160.000, Y  +661.396, Z    +0.000, E1    +6.484, E3 +175770.671}
SPL {X  -160.000, Y  +653.532, Z    +0.000, E1   +13.136, E3 +175774.791}
SPL {X  -160.000, Y  +631.927, Z    +0.000, E1   +26.832, E3 +175797.558}
SPL {X  -160.000, Y  +610.736, Z    +0.000, E1   +32.114, E3 +175840.227}
SPL {X  -160.000, Y  +605.907, Z    +0.000, E1   +32.114, E3 +175856.575}
SPL {X  -160.000, Y  +601.221, Z    +0.000, E1   +32.108, E3 +175872.443}
SPL {X  -160.000, Y  +596.433, Z    +0.000, E1   +32.120, E3 +175888.625}
SPL {X  -160.000, Y  +592.025, Z    +0.000, E1   +32.104, E3 +175903.550}
SPL {X  -160.000, Y  +587.734, Z    +0.000, E1   +32.110, E3 +175918.070}
SPL {X  -160.000, Y  +583.150, Z    +0.000, E1   +32.111, E3 +175933.597}
SPL {X  -160.000, Y  +579.063, Z    +0.000, E1   +32.085, E3 +175947.499}
SPL {X  -160.000, Y  +574.897, Z    +0.000, E1   +32.110, E3 +175961.550}
SPL {X  -160.000, Y  +570.471, Z    +0.000, E1   +32.093, E3 +175976.564}
SPL {X  -160.000, Y  +566.667, Z    +0.000, E1   +32.086, E3 +175989.479}
SPL {X  -160.000, Y  +562.434, Z    +0.000, E1   +32.097, E3 +176003.788}
SPL {X  -160.000, Y  +557.710, Z    +0.000, E1   +32.104, E3 +176019.772}
SPL {X  -160.000, Y  +553.479, Z    +0.000, E1   +32.081, E3 +176034.141}
SPL {X  -160.000, Y  +547.489, Z    +0.000, E1   +32.181, E3 +176054.260}
SPL {X  -160.000, Y  +541.554, Z    +0.000, E1   +32.092, E3 +176074.497}
SPL {X  -160.000, Y  +537.332, Z    +0.000, E1   +32.092, E3 +176088.794}
SPL {X  -160.000, Y  +533.113, Z    +0.000, E1   +32.090, E3 +176103.091}
SPL {X  -160.000, Y  +528.875, Z    +0.000, E1   +32.090, E3 +176117.434}
SPL {X  -160.000, Y  +524.453, Z    +0.000, E1   +32.104, E3 +176132.358}
SPL {X  -160.000, Y  +520.037, Z    +0.000, E1   +32.096, E3 +176147.300}
SPL {X  -160.000, Y  +514.030, Z    +0.000, E1   +32.182, E3 +176167.496}
SPL {X  -160.000, Y  +508.131, Z    +0.000, E1   +32.099, E3 +176187.601}
SPL {X  -160.000, Y  +504.077, Z    +0.000, E1   +32.094, E3 +176201.323}
SPL {X  -160.000, Y  +494.657, Z    +0.000, E1   +34.509, E3 +176216.186}
SPL {X  -160.000, Y  +491.565, Z    +0.000, E1   +33.823, E3 +176230.094}
SPL {X  -160.000, Y  +489.317, Z    +0.000, E1   +32.894, E3 +176243.438}
SPL {X  -160.000, Y  +486.958, Z    +0.000, E1   +31.703, E3 +176259.210}
SPL {X  -160.000, Y  +484.144, Z    +0.000, E1   +30.999, E3 +176273.633}
SPL {X  -160.000, Y  +479.156, Z    +0.000, E1   +31.035, E3 +176291.199}
SPL {X  -160.000, Y  +474.045, Z    +0.000, E1   +31.015, E3 +176309.291}
SPL {X  -160.000, Y  +468.999, Z    +0.000, E1   +31.021, E3 +176327.116}
SPL {X  -160.000, Y  +464.107, Z    +0.000, E1   +31.012, E3 +176344.416}
SPL {X  -160.000, Y  +459.262, Z    +0.000, E1   +31.016, E3 +176361.523}
SPL {X  -160.000, Y  +454.119, Z    +0.000, E1   +31.026, E3 +176379.672}
SPL {X  -160.000, Y  +448.874, Z    +0.000, E1   +31.019, E3 +176398.228}
SPL {X  -160.000, Y  +443.892, Z    +0.000, E1   +31.019, E3 +176415.816}
SPL {X  -160.000, Y  +438.782, Z    +0.000, E1   +31.022, E3 +176433.891}
SPL {X  -160.000, Y  +433.722, Z    +0.000, E1   +31.007, E3 +176451.835}
SPL {X  -160.000, Y  +428.980, Z    +0.000, E1   +31.004, E3 +176468.592}
SPL {X  -160.000, Y  +424.339, Z    +0.000, E1   +31.006, E3 +176484.966}
SPL {X  -160.000, Y  +419.231, Z    +0.000, E1   +31.030, E3 +176502.960}
SPL {X  -160.000, Y  +414.179, Z    +0.000, E1   +31.008, E3 +176520.857}
SPL {X  -160.000, Y  +409.416, Z    +0.000, E1   +31.023, E3 +176537.640}
SPL {X  -160.000, Y  +403.994, Z    +0.000, E1   +31.033, E3 +176556.796}
SPL {X  -160.000, Y  +399.052, Z    +0.000, E1   +31.010, E3 +176574.264}
SPL {X  -160.000, Y  +394.012, Z    +0.000, E1   +31.036, E3 +176592.052}
SPL {X  -159.999, Y  +388.376, Z    +0.000, E1   +31.028, E3 +176611.982}
SPL {X  -159.897, Y  +383.070, Z    +0.000, E1   +31.010, E3 +176630.820}
SPL {X  -159.656, Y  +378.313, Z    +0.000, E1   +30.961, E3 +176647.912}
SPL {X  -159.237, Y  +373.190, Z    +0.000, E1   +30.917, E3 +176666.412}
SPL {X  -158.628, Y  +367.891, Z    +0.000, E1   +30.812, E3 +176685.798}
SPL {X  -157.915, Y  +363.053, Z    +0.000, E1   +30.689, E3 +176703.665}
SPL {X  -157.216, Y  +359.084, Z    +0.000, E1   +30.550, E3 +176718.468}
SPL {X  -156.248, Y  +354.355, Z    +0.000, E1   +30.460, E3 +176736.080}
SPL {X  -155.629, Y  +351.657, Z    +0.000, E1   +25.972, E3 +176782.508}
ENDSPLINE

SPLINE
SPL {X  -156.240, Y  +354.319, Z    +0.000, E1   +23.538, E3 +176795.116}
SPL {X  -159.137, Y  +372.201, Z    +0.000, E1   +12.017, E3 +176824.953}
SPL {X  -159.858, Y  +382.069, Z    +0.000, E1    +5.945, E3 +176831.471}
SPL {X  -160.000, Y  +389.339, Z    +0.000, E1    +1.101, E3 +176834.633}
SPL {X  -160.000, Y  +395.749, Z    +0.000, E1    -3.722, E3 +176837.238}
SPL {X  -160.000, Y  +403.128, Z    +0.000, E1    -9.899, E3 +176840.543}
SPL {X  -160.000, Y  +411.609, Z    +0.000, E1   -16.851, E3 +176845.864}
SPL {X  -160.000, Y  +429.715, Z    +0.000, E1   -27.376, E3 +176865.227}
SPL {X  -160.000, Y  +449.791, Z    +0.000, E1   -32.145, E3 +176906.464}
SPL {X  -160.000, Y  +454.903, Z    +0.000, E1   -32.134, E3 +176923.768}
SPL {X  -160.000, Y  +460.041, Z    +0.000, E1   -32.144, E3 +176941.122}
SPL {X  -160.000, Y  +465.466, Z    +0.000, E1   -32.152, E3 +176959.440}
SPL {X  -160.000, Y  +471.112, Z    +0.000, E1   -32.154, E3 +176978.528}
SPL {X  -160.000, Y  +476.735, Z    +0.000, E1   -32.156, E3 +176997.519}
SPL {X  -160.000, Y  +482.675, Z    +0.000, E1   -32.169, E3 +177017.568}
SPL {X  -160.000, Y  +488.008, Z    +0.000, E1   -32.144, E3 +177035.614}
SPL {X  -160.000, Y  +493.245, Z    +0.000, E1   -32.159, E3 +177053.322}
SPL {X  -160.000, Y  +498.210, Z    +0.000, E1   -32.128, E3 +177070.157}
SPL {X  -160.000, Y  +503.407, Z    +0.000, E1   -32.165, E3 +177087.661}
SPL {X  -160.000, Y  +509.142, Z    +0.000, E1   -32.157, E3 +177107.056}
SPL {X  -160.000, Y  +514.696, Z    +0.000, E1   -32.156, E3 +177125.837}
SPL {X  -160.000, Y  +520.339, Z    +0.000, E1   -32.159, E3 +177144.909}
SPL {X  -160.000, Y  +525.825, Z    +0.000, E1   -32.148, E3 +177163.473}
SPL {X  -160.000, Y  +530.379, Z    +0.000, E1   -32.130, E3 +177178.901}
SPL {X  -160.000, Y  +535.020, Z    +0.000, E1   -32.146, E3 +177194.547}
SPL {X  -160.000, Y  +540.303, Z    +0.000, E1   -32.158, E3 +177212.372}
SPL {X  -160.000, Y  +545.740, Z    +0.000, E1   -32.155, E3 +177230.765}
SPL {X  -160.000, Y  +550.807, Z    +0.000, E1   -32.147, E3 +177247.887}
SPL {X  -160.000, Y  +555.841, Z    +0.000, E1   -32.148, E3 +177264.927}
SPL {X  -160.000, Y  +561.018, Z    +0.000, E1   -32.143, E3 +177282.456}
SPL {X  -160.000, Y  +566.466, Z    +0.000, E1   -32.153, E3 +177300.874}
SPL {X  -160.000, Y  +571.733, Z    +0.000, E1   -32.135, E3 +177318.710}
SPL {X  -160.000, Y  +576.943, Z    +0.000, E1   -32.148, E3 +177336.307}
SPL {X  -160.000, Y  +582.183, Z    +0.000, E1   -32.140, E3 +177354.032}
SPL {X  -160.000, Y  +587.036, Z    +0.000, E1   -32.141, E3 +177370.403}
SPL {X  -160.000, Y  +591.785, Z    +0.000, E1   -32.144, E3 +177386.426}
SPL {X  -160.000, Y  +596.962, Z    +0.000, E1   -32.161, E3 +177403.913}
SPL {X  -160.000, Y  +601.800, Z    +0.000, E1   -32.134, E3 +177420.310}
SPL {X  -160.000, Y  +606.611, Z    +0.000, E1   -32.156, E3 +177436.525}
SPL {X  -160.000, Y  +611.219, Z    +0.000, E1   -32.131, E3 +177452.138}
SPL {X  -160.000, Y  +616.331, Z    +0.000, E1   -32.174, E3 +177469.336}
SPL {X  -160.000, Y  +621.751, Z    +0.000, E1   -32.150, E3 +177487.678}
SPL {X  -160.000, Y  +626.312, Z    +0.000, E1   -32.145, E3 +177503.084}
SPL {X  -160.000, Y  +630.971, Z    +0.000, E1   -32.155, E3 +177518.812}
SPL {X  -160.000, Y  +635.550, Z    +0.000, E1   -32.137, E3 +177534.338}
SPL {X  -160.000, Y  +640.419, Z    +0.000, E1   -32.158, E3 +177550.776}
SPL {X  -160.000, Y  +645.749, Z    +0.000, E1   -32.151, E3 +177568.802}
SPL {X  -160.000, Y  +650.662, Z    +0.000, E1   -32.150, E3 +177585.373}
SPL {X  -160.000, Y  +655.372, Z    +0.000, E1   -32.145, E3 +177601.320}
SPL {X  -160.000, Y  +660.593, Z    +0.000, E1   -32.163, E3 +177618.937}
SPL {X  -160.000, Y  +665.836, Z    +0.000, E1   -32.154, E3 +177636.654}
SPL {X  -160.000, Y  +670.613, Z    +0.000, E1   -32.138, E3 +177652.864}
SPL {X  -159.954, Y  +675.336, Z    +0.000, E1   -32.135, E3 +177668.873}
SPL {X  -159.758, Y  +680.302, Z    +0.000, E1   -32.108, E3 +177685.887}
SPL {X  -159.416, Y  +685.158, Z    +0.000, E1   -32.039, E3 +177702.699}
SPL {X  -158.953, Y  +689.772, Z    +0.000, E1   -31.965, E3 +177718.798}
SPL {X  -158.363, Y  +694.328, Z    +0.000, E1   -31.871, E3 +177734.810}
SPL {X  -157.606, Y  +699.074, Z    +0.000, E1   -31.756, E3 +177751.654}
SPL {X  -156.791, Y  +703.384, Z    +0.000, E1   -31.607, E3 +177767.104}
SPL {X  -155.792, Y  +707.952, Z    +0.000, E1   -31.465, E3 +177783.550}
SPL {X  -155.149, Y  +710.598, Z    +0.000, E1   -26.183, E3 +177839.010}
ENDSPLINE

SPLINE
SPL {X  -158.679, Y  +692.020, Z    +0.000, E1   -14.212, E3 +177872.686}
SPL {X  -159.747, Y  +680.500, Z    +0.000, E1    -7.378, E3 +177881.064}
SPL {X  -160.000, Y  +671.618, Z    +0.000, E1    -1.592, E3 +177884.679}
SPL {X  -160.000, Y  +666.041, Z    +0.000, E1    +2.615, E3 +177886.645}
SPL {X  -160.000, Y  +661.396, Z    +0.000, E1    +6.484, E3 +177888.318}
SPL {X  -160.000, Y  +653.532, Z    +0.000, E1   +13.136, E3 +177892.438}
SPL {X  -160.000, Y  +631.927, Z    +0.000, E1   +26.832, E3 +177915.205}
SPL {X  -160.000, Y  +610.736, Z    +0.000, E1   +32.114, E3 +177957.874}
SPL {X  -160.000, Y  +605.907, Z    +0.000, E1   +32.114, E3 +177974.223}
SPL {X  -160.000, Y  +601.221, Z    +0.000, E1   +32.108, E3 +177990.090}
SPL {X  -160.000, Y  +596.433, Z    +0.000, E1   +32.120, E3 +178006.272}
SPL {X  -160.000, Y  +592.025, Z    +0.000, E1   +32.104, E3 +178021.197}
SPL {X  -160.000, Y  +587.734, Z    +0.000, E1   +32.110, E3 +178035.717}
SPL {X  -160.000, Y  +583.150, Z    +0.000, E1   +32.111, E3 +178051.245}
SPL {X  -160.000, Y  +579.063, Z    +0.000, E1   +32.085, E3 +178065.146}
SPL {X  -160.000, Y  +574.897, Z    +0.000, E1   +32.110, E3 +178079.197}
SPL {X  -160.000, Y  +570.471, Z    +0.000, E1   +32.093, E3 +178094.212}
SPL {X  -160.000, Y  +566.667, Z    +0.000, E1   +32.086, E3 +178107.126}
SPL {X  -160.000, Y  +562.434, Z    +0.000, E1   +32.097, E3 +178121.436}
SPL {X  -160.000, Y  +557.710, Z    +0.000, E1   +32.104, E3 +178137.419}
SPL {X  -160.000, Y  +553.479, Z    +0.000, E1   +32.081, E3 +178151.788}
SPL {X  -160.000, Y  +547.489, Z    +0.000, E1   +32.181, E3 +178171.907}
SPL {X  -160.000, Y  +541.554, Z    +0.000, E1   +32.092, E3 +178192.144}
SPL {X  -160.000, Y  +537.332, Z    +0.000, E1   +32.092, E3 +178206.441}
SPL {X  -160.000, Y  +533.113, Z    +0.000, E1   +32.090, E3 +178220.738}
SPL {X  -160.000, Y  +528.875, Z    +0.000, E1   +32.090, E3 +178235.081}
SPL {X  -160.000, Y  +524.453, Z    +0.000, E1   +32.104, E3 +178250.005}
SPL {X  -160.000, Y  +520.037, Z    +0.000, E1   +32.096, E3 +178264.947}
SPL {X  -160.000, Y  +514.030, Z    +0.000, E1   +32.182, E3 +178285.143}
SPL {X  -160.000, Y  +508.131, Z    +0.000, E1   +32.099, E3 +178305.248}
SPL {X  -160.000, Y  +504.077, Z    +0.000, E1   +32.094, E3 +178318.971}
SPL {X  -160.000, Y  +494.657, Z    +0.000, E1   +34.509, E3 +178333.834}
SPL {X  -160.000, Y  +491.565, Z    +0.000, E1   +33.823, E3 +178347.741}
SPL {X  -160.000, Y  +489.317, Z    +0.000, E1   +32.894, E3 +178361.086}
SPL {X  -160.000, Y  +486.958, Z    +0.000, E1   +31.703, E3 +178376.857}
SPL {X  -160.000, Y  +484.144, Z    +0.000, E1   +30.999, E3 +178391.280}
SPL {X  -160.000, Y  +479.156, Z    +0.000, E1   +31.035, E3 +178408.846}
SPL {X  -160.000, Y  +474.045, Z    +0.000, E1   +31.015, E3 +178426.938}
SPL {X  -160.000, Y  +468.999, Z    +0.000, E1   +31.021, E3 +178444.763}
SPL {X  -160.000, Y  +464.107, Z    +0.000, E1   +31.012, E3 +178462.063}
SPL {X  -160.000, Y  +459.262, Z    +0.000, E1   +31.016, E3 +178479.170}
SPL {X  -160.000, Y  +454.119, Z    +0.000, E1   +31.026, E3 +178497.320}
SPL {X  -160.000, Y  +448.874, Z    +0.000, E1   +31.019, E3 +178515.876}
SPL {X  -160.000, Y  +443.892, Z    +0.000, E1   +31.019, E3 +178533.464}
SPL {X  -160.000, Y  +438.782, Z    +0.000, E1   +31.022, E3 +178551.538}
SPL {X  -160.000, Y  +433.722, Z    +0.000, E1   +31.007, E3 +178569.482}
SPL {X  -160.000, Y  +428.980, Z    +0.000, E1   +31.004, E3 +178586.239}
SPL {X  -160.000, Y  +424.339, Z    +0.000, E1   +31.006, E3 +178602.613}
SPL {X  -160.000, Y  +419.231, Z    +0.000, E1   +31.030, E3 +178620.607}
SPL {X  -160.000, Y  +414.179, Z    +0.000, E1   +31.008, E3 +178638.504}
SPL {X  -160.000, Y  +409.416, Z    +0.000, E1   +31.023, E3 +178655.287}
SPL {X  -160.000, Y  +403.994, Z    +0.000, E1   +31.033, E3 +178674.443}
SPL {X  -160.000, Y  +399.052, Z    +0.000, E1   +31.010, E3 +178691.911}
SPL {X  -160.000, Y  +394.012, Z    +0.000, E1   +31.036, E3 +178709.700}
SPL {X  -159.999, Y  +388.376, Z    +0.000, E1   +31.028, E3 +178729.629}
SPL {X  -159.897, Y  +383.070, Z    +0.000, E1   +31.010, E3 +178748.467}
SPL {X  -159.656, Y  +378.313, Z    +0.000, E1   +30.961, E3 +178765.560}
SPL {X  -159.237, Y  +373.190, Z    +0.000, E1   +30.917, E3 +178784.060}
SPL {X  -158.628, Y  +367.891, Z    +0.000, E1   +30.812, E3 +178803.445}
SPL {X  -157.915, Y  +363.053, Z    +0.000, E1   +30.689, E3 +178821.312}
SPL {X  -157.216, Y  +359.084, Z    +0.000, E1   +30.550, E3 +178836.115}
SPL {X  -156.248, Y  +354.355, Z    +0.000, E1   +30.460, E3 +178853.727}
SPL {X  -155.629, Y  +351.657, Z    +0.000, E1   +25.972, E3 +178900.156}
ENDSPLINE

SPLINE
SPL {X  -156.240, Y  +354.319, Z    +0.000, E1   +23.538, E3 +178912.763}
SPL {X  -159.137, Y  +372.201, Z    +0.000, E1   +12.017, E3 +178942.601}
SPL {X  -159.858, Y  +382.069, Z    +0.000, E1    +5.945, E3 +178949.118}
SPL {X  -160.000, Y  +389.339, Z    +0.000, E1    +1.101, E3 +178952.280}
SPL {X  -160.000, Y  +395.749, Z    +0.000, E1    -3.722, E3 +178954.886}
SPL {X  -160.000, Y  +403.128, Z    +0.000, E1    -9.899, E3 +178958.190}
SPL {X  -160.000, Y  +411.609, Z    +0.000, E1   -16.851, E3 +178963.511}
SPL {X  -160.000, Y  +429.715, Z    +0.000, E1   -27.376, E3 +178982.874}
SPL {X  -160.000, Y  +449.791, Z    +0.000, E1   -32.145, E3 +179024.111}
SPL {X  -160.000, Y  +454.903, Z    +0.000, E1   -32.134, E3 +179041.416}
SPL {X  -160.000, Y  +460.041, Z    +0.000, E1   -32.144, E3 +179058.769}
SPL {X  -160.000, Y  +465.466, Z    +0.000, E1   -32.152, E3 +179077.087}
SPL {X  -160.000, Y  +471.112, Z    +0.000, E1   -32.154, E3 +179096.175}
SPL {X  -160.000, Y  +476.735, Z    +0.000, E1   -32.156, E3 +179115.166}
SPL {X  -160.000, Y  +482.675, Z    +0.000, E1   -32.169, E3 +179135.215}
SPL {X  -160.000, Y  +488.008, Z    +0.000, E1   -32.144, E3 +179153.261}
SPL {X  -160.000, Y  +493.245, Z    +0.000, E1   -32.159, E3 +179170.970}
SPL {X  -160.000, Y  +498.210, Z    +0.000, E1   -32.128, E3 +179187.804}
SPL {X  -160.000, Y  +503.407, Z    +0.000, E1   -32.165, E3 +179205.308}
SPL {X  -160.000, Y  +509.142, Z    +0.000, E1   -32.157, E3 +179224.704}
SPL {X  -160.000, Y  +514.696, Z    +0.000, E1   -32.156, E3 +179243.484}
SPL {X  -160.000, Y  +520.339, Z    +0.000, E1   -32.159, E3 +179262.556}
SPL {X  -160.000, Y  +525.825, Z    +0.000, E1   -32.148, E3 +179281.120}
SPL {X  -160.000, Y  +530.379, Z    +0.000, E1   -32.130, E3 +179296.548}
SPL {X  -160.000, Y  +535.020, Z    +0.000, E1   -32.146, E3 +179312.194}
SPL {X  -160.000, Y  +540.303, Z    +0.000, E1   -32.158, E3 +179330.019}
SPL {X  -160.000, Y  +545.740, Z    +0.000, E1   -32.155, E3 +179348.412}
SPL {X  -160.000, Y  +550.807, Z    +0.000, E1   -32.147, E3 +179365.535}
SPL {X  -160.000, Y  +555.841, Z    +0.000, E1   -32.148, E3 +179382.574}
SPL {X  -160.000, Y  +561.018, Z    +0.000, E1   -32.143, E3 +179400.103}
SPL {X  -160.000, Y  +566.466, Z    +0.000, E1   -32.153, E3 +179418.521}
SPL {X  -160.000, Y  +571.733, Z    +0.000, E1   -32.135, E3 +179436.358}
SPL {X  -160.000, Y  +576.943, Z    +0.000, E1   -32.148, E3 +179453.954}
SPL {X  -160.000, Y  +582.183, Z    +0.000, E1   -32.140, E3 +179471.679}
SPL {X  -160.000, Y  +587.036, Z    +0.000, E1   -32.141, E3 +179488.050}
SPL {X  -160.000, Y  +591.785, Z    +0.000, E1   -32.144, E3 +179504.074}
SPL {X  -160.000, Y  +596.962, Z    +0.000, E1   -32.161, E3 +179521.560}
SPL {X  -160.000, Y  +601.800, Z    +0.000, E1   -32.134, E3 +179537.957}
SPL {X  -160.000, Y  +606.611, Z    +0.000, E1   -32.156, E3 +179554.172}
SPL {X  -160.000, Y  +611.219, Z    +0.000, E1   -32.131, E3 +179569.785}
SPL {X  -160.000, Y  +616.331, Z    +0.000, E1   -32.174, E3 +179586.983}
SPL {X  -160.000, Y  +621.751, Z    +0.000, E1   -32.150, E3 +179605.326}
SPL {X  -160.000, Y  +626.312, Z    +0.000, E1   -32.145, E3 +179620.731}
SPL {X  -160.000, Y  +630.971, Z    +0.000, E1   -32.155, E3 +179636.460}
SPL {X  -160.000, Y  +635.550, Z    +0.000, E1   -32.137, E3 +179651.985}
SPL {X  -160.000, Y  +640.419, Z    +0.000, E1   -32.158, E3 +179668.423}
SPL {X  -160.000, Y  +645.749, Z    +0.000, E1   -32.151, E3 +179686.449}
SPL {X  -160.000, Y  +650.662, Z    +0.000, E1   -32.150, E3 +179703.020}
SPL {X  -160.000, Y  +655.372, Z    +0.000, E1   -32.145, E3 +179718.967}
SPL {X  -160.000, Y  +660.593, Z    +0.000, E1   -32.163, E3 +179736.585}
SPL {X  -160.000, Y  +665.836, Z    +0.000, E1   -32.154, E3 +179754.301}
SPL {X  -160.000, Y  +670.613, Z    +0.000, E1   -32.138, E3 +179770.512}
SPL {X  -159.954, Y  +675.336, Z    +0.000, E1   -32.135, E3 +179786.520}
SPL {X  -159.758, Y  +680.302, Z    +0.000, E1   -32.108, E3 +179803.535}
SPL {X  -159.416, Y  +685.158, Z    +0.000, E1   -32.039, E3 +179820.346}
SPL {X  -158.953, Y  +689.772, Z    +0.000, E1   -31.965, E3 +179836.445}
SPL {X  -158.363, Y  +694.328, Z    +0.000, E1   -31.871, E3 +179852.458}
SPL {X  -157.606, Y  +699.074, Z    +0.000, E1   -31.756, E3 +179869.301}
SPL {X  -156.791, Y  +703.384, Z    +0.000, E1   -31.607, E3 +179884.751}
SPL {X  -155.792, Y  +707.952, Z    +0.000, E1   -31.465, E3 +179901.198}
SPL {X  -155.149, Y  +710.598, Z    +0.000, E1   -26.183, E3 +179956.657}
ENDSPLINE

